  MoveL 5922 to (-205.95, 106.69, -39.37) mm, rotated rx -180 ry 0 rz 0.01 deg; joints [32.683, -45.289, 105.651, -143.751, 66, 164.377]
  MoveL 5923 to (-200.36, 103.18, -39.61) mm, rotated rx 180 ry 0 rz 0.01 deg; joints [32.686, -45.553, 106.254, -143.837, 66.275, 164.595]
  MoveL 5924 to (-194.9, 106.89, -39.86) mm, rotated rx 180 ry 0 rz 0.01 deg; joints [32.922, -45.653, 106.489, -143.624, 66.452, 164.581]
  MoveL 5925 to (-196.11, 113.38, -40.1) mm, rotated rx -180 ry 0 rz 0.01 deg; joints [33.109, -45.453, 106.072, -143.373, 66.332, 164.36]
  MoveL 5926 to (-202.54, 114.87, -40.35) mm, rotated rx 180 ry 0 rz 0.01 deg; joints [33.021, -45.178, 105.502, -143.387, 66.069, 164.205]
  MoveL 5927 to (-206.49, 109.57, -40.59) mm, rotated rx 180 ry 0 rz 0.01 deg; joints [32.766, -45.142, 105.46, -143.652, 65.99, 164.313]
  MoveL 5928 to (-203.21, 103.84, -40.83) mm, rotated rx 180 ry 0 rz 0.01 deg; joints [32.648, -45.372, 105.996, -143.856, 66.202, 164.561]
  MoveL 5929 to (-196.65, 104.54, -41.08) mm, rotated rx -180 ry 0 rz 0.01 deg; joints [32.809, -45.577, 106.465, -143.756, 66.461, 164.662]
  MoveL 5930 to (-194.66, 110.84, -41.32) mm, rotated rx 180 ry 0 rz 0.01 deg; joints [33.057, -45.496, 106.304, -143.476, 66.469, 164.505]
  MoveL 5931 to (-199.63, 115.18, -41.57) mm, rotated rx -180 ry 0 rz 0.01 deg; joints [33.093, -45.21, 105.704, -143.357, 66.227, 164.285]
  MoveL 5932 to (-205.6, 112.37, -41.81) mm, rotated rx -180 ry 0 rz 0.01 deg; joints [32.876, -45.046, 105.383, -143.542, 66.037, 164.276]
  MoveL 5933 to (-205.42, 105.77, -42.05) mm, rotated rx 180 ry 0 rz 0.01 deg; joints [32.666, -45.186, 105.724, -143.815, 66.137, 164.498]
  MoveL 5934 to (-199.3, 103.29, -42.3) mm, rotated rx 180 ry 0 rz 0.01 deg; joints [32.713, -45.445, 106.317, -143.852, 66.42, 164.693]
  MoveL 5935 to (-194.57, 107.91, -42.54) mm, rotated rx 180 ry 0 rz 0.01 deg; joints [32.964, -45.498, 106.449, -143.611, 66.557, 164.637]
  MoveL 5936 to (-196.91, 114.08, -42.79) mm, rotated rx 180 ry 0 rz 0.01 deg; joints [33.116, -45.266, 105.962, -143.386, 66.396, 164.406]
  MoveL 5937 to (-203.51, 114.42, -43.03) mm, rotated rx 180 ry 0 rz 0.01 deg; joints [32.988, -45.011, 105.436, -143.449, 66.141, 164.286]
  MoveL 5938 to (-206.46, 108.51, -43.27) mm, rotated rx 180 ry 0 rz 0.01 deg; joints [32.734, -45.024, 105.501, -143.728, 66.109, 164.43]
  MoveL 5939 to (-202.22, 103.44, -43.52) mm, rotated rx 180 ry 0 rz 0.01 deg; joints [32.657, -45.273, 106.078, -143.893, 66.351, 164.674]
  MoveL 5940 to (-195.88, 105.28, -43.76) mm, rotated rx -180 ry 0 rz 0.01 deg; joints [32.851, -45.444, 106.472, -143.748, 66.587, 164.735]
  MoveL 5941 to (-195.03, 111.83, -44.01) mm, rotated rx 180 ry 0 rz 0.01 deg; joints [33.083, -45.317, 106.211, -143.472, 66.546, 164.549]
  MoveL 5942 to (-200.69, 115.24, -44.25) mm, rotated rx 180 ry 0 rz 0.01 deg; joints [33.074, -45.028, 105.605, -143.399, 66.288, 164.347]
  MoveL 5943 to (-206.08, 111.41, -44.49) mm, rotated rx 180 ry 0 rz 0.01 deg; joints [32.837, -44.908, 105.38, -143.619, 66.134, 164.381]
  MoveL 5944 to (-204.74, 104.95, -44.74) mm, rotated rx -180 ry 0 rz 0.01 deg; joints [32.655, -45.085, 105.803, -143.873, 66.279, 164.619]
  MoveL 5945 to (-198.27, 103.59, -44.98) mm, rotated rx 180 ry 0 rz 0.01 deg; joints [32.746, -45.331, 106.366, -143.86, 66.562, 164.784]
  MoveL 5946 to (-194.44, 108.96, -45.23) mm, rotated rx 180 ry 0 rz 0.01 deg; joints [33.003, -45.335, 106.393, -143.597, 66.654, 164.689]
  MoveL 5947 to (-197.83, 114.63, -45.47) mm, rotated rx 180 ry 0 rz 0.01 deg; joints [33.116, -45.078, 105.849, -143.406, 66.456, 164.456]
  MoveL 5948 to (-204.38, 113.8, -45.71) mm, rotated rx 180 ry 0 rz 0.01 deg; joints [32.951, -44.851, 105.385, -143.516, 66.217, 164.372]
  MoveL 5949 to (-206.24, 107.46, -45.96) mm, rotated rx 180 ry 0 rz 0.01 deg; joints [32.706, -44.912, 105.555, -143.801, 66.235, 164.549]
  MoveL 5950 to (-201.18, 103.22, -46.2) mm, rotated rx 180 ry 0 rz 0.01 deg; joints [32.673, -45.171, 106.154, -143.922, 66.499, 164.782]
  MoveL 5951 to (-195.26, 106.15, -46.45) mm, rotated rx -180 ry 0 rz 0.01 deg; joints [32.894, -45.302, 106.462, -143.737, 66.705, 164.801]
  MoveL 5952 to (-195.58, 112.75, -46.69) mm, rotated rx 180 ry 0 rz 0.01 deg; joints [33.103, -45.133, 106.109, -143.472, 66.616, 164.594]
  MoveL 5953 to (-201.75, 115.1, -46.93) mm, rotated rx -180 ry 0 rz 0.01 deg; joints [33.049, -44.85, 105.516, -143.448, 66.352, 164.415]
  MoveL 5954 to (-206.38, 110.39, -47.18) mm, rotated rx -180 ry 0 rz 0.01 deg; joints [32.799, -44.777, 105.392, -143.696, 66.238, 164.49]
  MoveL 5955 to (-203.92, 104.26, -47.42) mm, rotated rx 180 ry 0 rz 0.01 deg; joints [32.651, -44.986, 105.885, -143.924, 66.425, 164.737]
  MoveL 5956 to (-197.32, 104.06, -47.67) mm, rotated rx 180 ry 0 rz 0.01 deg; joints [32.783, -45.21, 106.401, -143.861, 66.698, 164.868]
  MoveL 5957 to (-194.49, 110.03, -47.91) mm, rotated rx -180 ry 0 rz 0.01 deg; joints [33.038, -45.166, 106.321, -143.585, 66.742, 164.737]
  MoveL 5958 to (-198.82, 115.01, -48.15) mm, rotated rx -180 ry 0 rz 0.01 deg; joints [33.109, -44.891, 105.739, -143.433, 66.516, 164.508]
  MoveL 5959 to (-205.13, 113.04, -48.4) mm, rotated rx -180 ry 0 rz 0.01 deg; joints [32.912, -44.698, 105.35, -143.588, 66.301, 164.466]
  MoveL 5960 to (-205.84, 106.47, -48.64) mm, rotated rx -180 ry 0 rz 0.01 deg; joints [32.683, -44.804, 105.62, -143.869, 66.367, 164.67]
  MoveL 5961 to (-200.11, 103.19, -48.89) mm, rotated rx -180 ry 0 rz 0.01 deg; joints [32.696, -45.065, 106.222, -143.943, 66.646, 164.884]
  MoveL 5962 to (-194.81, 107.12, -49.13) mm, rotated rx -180 ry 0 rz 0.01 deg; joints [32.937, -45.153, 106.434, -143.723, 66.815, 164.861]
  MoveL 5963 to (-196.28, 113.55, -49.38) mm, rotated rx 180 ry 0 rz 0.01 deg; joints [33.116, -44.947, 106, -143.478, 66.682, 164.638]
  MoveL 5964 to (-202.77, 114.78, -49.62) mm, rotated rx 180 ry 0 rz 0.01 deg; joints [33.019, -44.678, 105.438, -143.504, 66.418, 164.49]
  MoveL 5965 to (-206.5, 109.33, -49.86) mm, rotated rx -180 ry 0 rz 0.01 deg; joints [32.763, -44.653, 105.421, -143.773, 66.351, 164.604]
  MoveL 5966 to (-202.99, 103.73, -50.11) mm, rotated rx -180 ry 0 rz 0.01 deg; joints [32.654, -44.886, 105.967, -143.967, 66.572, 164.852]
  MoveL 5967 to (-196.46, 104.7, -50.35) mm, rotated rx 180 ry 0 rz 0.01 deg; joints [32.824, -45.082, 106.42, -143.856, 66.828, 164.946]
  MoveL 5968 to (-194.73, 111.07, -50.6) mm, rotated rx -180 ry 0 rz 0.01 deg; joints [33.069, -44.991, 106.235, -143.577, 66.823, 164.782]
  MoveL 5969 to (-199.87, 115.21, -50.84) mm, rotated rx -180 ry 0 rz 0.01 deg; joints [33.094, -44.706, 105.633, -143.468, 66.575, 164.565]
  MoveL 5970 to (-205.73, 112.16, -51.08) mm, rotated rx -180 ry 0 rz 0.01 deg; joints [32.872, -44.553, 105.332, -143.662, 66.391, 164.565]
  MoveL 5971 to (-205.28, 105.57, -51.33) mm, rotated rx -180 ry 0 rz 0.01 deg; joints [32.667, -44.7, 105.692, -143.931, 66.505, 164.79]
  MoveL 5972 to (-199.06, 103.34, -51.57) mm, rotated rx -180 ry 0 rz 0.01 deg; joints [32.725, -44.954, 106.28, -143.955, 66.791, 164.979]
  MoveL 5973 to (-194.53, 108.15, -51.82) mm, rotated rx -180 ry 0 rz 0.01 deg; joints [32.978, -44.996, 106.389, -143.708, 66.916, 164.916]
  MoveL 5974 to (-197.11, 114.22, -52.06) mm, rotated rx 180 ry 0 rz 0.01 deg; joints [33.121, -44.759, 105.886, -143.492, 66.744, 164.684]
  MoveL 5975 to (-203.72, 114.29, -52.3) mm, rotated rx 180 ry 0 rz 0.01 deg; joints [32.984, -44.512, 105.374, -143.566, 66.49, 164.57]
  MoveL 5976 to (-206.42, 108.27, -52.55) mm, rotated rx 180 ry 0 rz 0.01 deg; joints [32.732, -44.536, 105.463, -143.847, 66.471, 164.721]
  MoveL 5977 to (-201.99, 103.37, -52.79) mm, rotated rx 180 ry 0 rz 0.01 deg; joints [32.665, -44.785, 106.046, -144.001, 66.721, 164.963]
  MoveL 5978 to (-195.73, 105.47, -53.04) mm, rotated rx 180 ry 0 rz 0.01 deg; joints [32.866, -44.946, 106.421, -143.846, 66.951, 165.016]
  MoveL 5979 to (-195.14, 112.05, -53.28) mm, rotated rx 180 ry 0 rz 0.01 deg; joints [33.093, -44.81, 106.138, -143.572, 66.897, 164.826]
  MoveL 5980 to (-200.94, 115.22, -53.52) mm, rotated rx 180 ry 0 rz 0.01 deg; joints [33.074, -44.525, 105.534, -143.511, 66.635, 164.628]
  MoveL 5981 to (-206.16, 111.18, -53.77) mm, rotated rx -180 ry 0 rz 0.01 deg; joints [32.833, -44.416, 105.33, -143.738, 66.489, 164.669]
  MoveL 5982 to (-204.56, 104.78, -54.01) mm, rotated rx 180 ry 0 rz 0.01 deg; joints [32.658, -44.599, 105.77, -143.986, 66.647, 164.909]
  MoveL 5983 to (-198.05, 103.68, -54.26) mm, rotated rx 180 ry 0 rz 0.01 deg; joints [32.759, -44.838, 106.324, -143.96, 66.93, 165.068]
  MoveL 5984 to (-194.43, 109.21, -54.5) mm, rotated rx 180 ry 0 rz 0.01 deg; joints [33.016, -44.831, 106.326, -143.694, 67.01, 164.966]
  MoveC 5985 to (-196.76, 111.53, -54.5) mm, rotated rx 180 ry 0 rz 0.01 deg; joints [33.043, -44.7, 106.033, -143.626, 66.887, 164.85] to (-199.08, 109.21, -54.5) mm, rotated rx -180 ry 0 rz 0.01 deg; joints [32.918, -44.669, 105.97, -143.748, 66.826, 164.882]
  MoveC 5986 to (-196.76, 106.88, -54.5) mm, rotated rx -180 ry 0 rz 0.01 deg; joints [32.891, -44.801, 106.264, -143.817, 66.949, 164.997] to (-194.43, 109.21, -54.5) mm, rotated rx -180 ry 0 rz 0.01 deg; joints [33.016, -44.831, 106.326, -143.694, 67.01, 164.966]
  MoveC 5987 to (-193.87, 111.26, -54.5) mm, rotated rx 180 ry 0 rz 0.01 deg; joints [33.095, -44.806, 106.268, -143.604, 67.005, 164.911] to (-192.35, 112.73, -54.5) mm, rotated rx -180 ry 0 rz 0.01 deg; joints [33.176, -44.827, 106.311, -143.526, 67.046, 164.892]
  MoveC 5988 to (-191.13, 114.78, -54.5) mm, rotated rx -180 ry 0 rz 0.01 deg; joints [33.268, -44.825, 106.301, -143.428, 67.066, 164.849] to (-192.33, 116.83, -54.5) mm, rotated rx 180 ry 0 rz 0.01 deg; joints [33.309, -44.738, 106.107, -143.358, 66.992, 164.762]
  MoveC 5989 to (-193.08, 117.28, -54.5) mm, rotated rx -180 ry 0 rz 0.01 deg; joints [33.308, -44.702, 106.027, -143.348, 66.956, 164.734] to (-193.81, 117.76, -54.5) mm, rotated rx 180 ry 0 rz 0.01 deg; joints [33.308, -44.666, 105.947, -143.337, 66.921, 164.705]
  MoveC 5990 to (-196.76, 118.7, -54.5) mm, rotated rx 180 ry 0 rz 0.01 deg; joints [33.275, -44.542, 105.675, -143.332, 66.792, 164.622] to (-199.7, 117.76, -54.5) mm, rotated rx 180 ry 0 rz 0.01 deg; joints [33.183, -44.46, 105.496, -143.404, 66.688, 164.599]
  MoveC 5991 to (-201.1, 116.87, -54.5) mm, rotated rx 180 ry 0 rz 0.01 deg; joints [33.124, -44.43, 105.432, -143.456, 66.644, 164.602] to (-202.59, 116.12, -54.5) mm, rotated rx -180 ry 0 rz 0.01 deg; joints [33.069, -44.394, 105.355, -143.504, 66.595, 164.599]
  MoveC 5992 to (-204.95, 114.01, -54.5) mm, rotated rx 180 ry 0 rz 0.01 deg; joints [32.951, -44.358, 105.279, -143.617, 66.529, 164.623] to (-205.64, 110.92, -54.5) mm, rotated rx -180 ry 0 rz 0.01 deg; joints [32.836, -44.401, 105.38, -143.751, 66.542, 164.709]
  MoveC 5993 to (-205.56, 109.27, -54.5) mm, rotated rx -180 ry 0 rz 0.01 deg; joints [32.784, -44.44, 105.467, -143.819, 66.567, 164.763] to (-205.65, 107.61, -54.5) mm, rotated rx 180 ry 0 rz 0.01 deg; joints [32.728, -44.473, 105.543, -143.888, 66.585, 164.814]
  MoveC 5994 to (-205, 104.51, -54.5) mm, rotated rx 180 ry 0 rz 0.01 deg; joints [32.64, -44.563, 105.747, -144.008, 66.652, 164.924] to (-202.66, 102.37, -54.5) mm, rotated rx -180 ry 0 rz 0.01 deg; joints [32.619, -44.691, 106.032, -144.07, 66.773, 165.034]
  MoveC 5995 to (-201.23, 101.62, -54.5) mm, rotated rx -180 ry 0 rz 0.01 deg; joints [32.625, -44.758, 106.18, -144.084, 66.841, 165.083] to (-199.87, 100.74, -54.5) mm, rotated rx -180 ry 0 rz 0.01 deg; joints [32.624, -44.824, 106.328, -144.105, 66.906, 165.135]
  MoveC 5996 to (-196.86, 99.74, -54.5) mm, rotated rx -180 ry 0 rz 0.01 deg; joints [32.655, -44.951, 106.608, -144.112, 67.039, 165.22] to (-193.81, 100.62, -54.5) mm, rotated rx -180 ry 0 rz 0.01 deg; joints [32.748, -45.038, 106.797, -144.04, 67.148, 165.247]
  MoveC 5997 to (-193.08, 101.1, -54.5) mm, rotated rx 180 ry 0 rz 0.01 deg; joints [32.779, -45.053, 106.83, -144.011, 67.171, 165.245] to (-192.33, 101.56, -54.5) mm, rotated rx -180 ry 0 rz 0.01 deg; joints [32.81, -45.069, 106.864, -143.984, 67.194, 165.244]
  MoveC 5998 to (-191.57, 102, -54.5) mm, rotated rx -180 ry 0 rz 0.01 deg; joints [32.841, -45.086, 106.901, -143.957, 67.219, 165.244] to (-190.79, 102.39, -54.5) mm, rotated rx -180 ry 0 rz 0.01 deg; joints [32.87, -45.105, 106.941, -143.931, 67.244, 165.245]
  MoveC 5999 to (-188.5, 104.54, -54.5) mm, rotated rx -180 ry 0 rz 0.01 deg; joints [32.99, -45.138, 107.011, -143.816, 67.306, 165.219] to (-187.86, 107.61, -54.5) mm, rotated rx -180 ry 0 rz 0.01 deg; joints [33.104, -45.094, 106.907, -143.682, 67.291, 165.134]
  MoveC 6000 to (-187.95, 109.27, -54.5) mm, rotated rx 180 ry 0 rz 0.01 deg; joints [33.156, -45.055, 106.819, -143.616, 67.265, 165.08] to (-187.87, 110.92, -54.5) mm, rotated rx 180 ry 0 rz 0.01 deg; joints [33.212, -45.022, 106.742, -143.547, 67.246, 165.029]
  MoveC 6001 to (-188.56, 114.01, -54.5) mm, rotated rx 180 ry 0 rz 0.01 deg; joints [33.298, -44.931, 106.535, -143.429, 67.178, 164.919] to (-190.92, 116.12, -54.5) mm, rotated rx 180 ry 0 rz 0.01 deg; joints [33.316, -44.802, 106.25, -143.37, 67.057, 164.81]
  MoveC 6002 to (-191.64, 116.46, -54.5) mm, rotated rx 180 ry 0 rz 0.01 deg; joints [33.312, -44.77, 106.179, -143.365, 67.024, 164.786] to (-192.33, 116.83, -54.5) mm, rotated rx 180 ry 0 rz 0.01 deg; joints [33.309, -44.738, 106.107, -143.358, 66.992, 164.762]
  MoveL 6003 to (-192.94, 116.99, -54.33) mm, rotated rx 180 ry 0 rz 0.01 deg; joints [33.301, -44.722, 106.054, -143.356, 66.959, 164.741]
  MoveL 6004 to (-193.39, 116.91, -53.87) mm, rotated rx -180 ry 0 rz 0.01 deg; joints [33.289, -44.733, 106.026, -143.359, 66.924, 164.721]
  MoveL 6005 to (-193.55, 116.84, -53.23) mm, rotated rx 180 ry 0 rz 0.01 deg; joints [33.283, -44.764, 106.021, -143.357, 66.895, 164.701]
  Set speed (500.0 mm/s)
  MoveL 6006 to (-193.55, 116.84, 11) mm, rotated rx 180 ry 0 rz 0.01 deg; joints [33.247, -48.144, 106.249, -142.533, 64.368, 162.631]
  Set speed (500.0 mm/s)
  MoveL 6007 to (-195.99, 9.53, 11) mm, rotated rx -180 ry 0 rz 0.01 deg; joints [29.569, -50.402, 111.086, -147.114, 65.397, 165.962]
  Set speed (500.0 mm/s)
  MoveL 6008 to (-195.99, 9.53, -32.73) mm, rotated rx 180 ry 0 rz 0.01 deg; joints [29.597, -48.003, 110.965, -147.623, 67.321, 167.29]
  Set speed (100.0 mm/s)
  MoveL 6009 to (-196.15, 9.55, -33.35) mm, rotated rx 180 ry 0 rz 0.01 deg; joints [29.595, -47.963, 110.949, -147.63, 67.342, 167.305]
  MoveL 6010 to (-196.6, 9.58, -33.82) mm, rotated rx 180 ry 0 rz 0.01 deg; joints [29.587, -47.921, 110.911, -147.639, 67.344, 167.311]
  MoveL 6011 to (-197.22, 9.56, -34) mm, rotated rx -180 ry 0 rz 0.01 deg; joints [29.574, -47.889, 110.864, -147.649, 67.327, 167.307]
  MoveL 6012 to (-202.45, 5.54, -34.24) mm, rotated rx -180 ry 0 rz 0.01 deg; joints [29.33, -47.766, 110.634, -147.882, 67.177, 167.348]
  MoveL 6013 to (-200.86, -0.87, -34.49) mm, rotated rx 180 ry 0 rz 0.01 deg; joints [29.136, -47.93, 111.031, -148.138, 67.329, 167.563]
  MoveL 6014 to (-194.35, -1.99, -34.73) mm, rotated rx 180 ry 0 rz 0.01 deg; joints [29.225, -48.167, 111.578, -148.112, 67.613, 167.703]
  MoveL 6015 to (-190.73, 3.53, -34.98) mm, rotated rx 180 ry 0 rz 0.01 deg; joints [29.492, -48.177, 111.617, -147.838, 67.701, 167.61]
  MoveL 6016 to (-194.33, 9.07, -35.22) mm, rotated rx 180 ry 0 rz 0.01 deg; joints [29.615, -47.932, 111.101, -147.649, 67.501, 167.403]
  MoveL 6017 to (-200.84, 7.98, -35.46) mm, rotated rx -180 ry 0 rz 0.01 deg; joints [29.448, -47.709, 110.646, -147.773, 67.265, 167.338]
  MoveL 6018 to (-202.46, 1.58, -35.71) mm, rotated rx -180 ry 0 rz 0.01 deg; joints [29.192, -47.759, 110.797, -148.066, 67.288, 167.503]
  MoveL 6019 to (-197.25, -2.47, -35.95) mm, rotated rx 180 ry 0 rz 0.01 deg; joints [29.152, -48.006, 111.371, -148.179, 67.557, 167.707]
  MoveL 6020 to (-191.44, 0.69, -36.2) mm, rotated rx 180 ry 0 rz 0.01 deg; joints [29.378, -48.137, 111.679, -147.98, 67.76, 167.715]
  MoveL 6021 to (-192.01, 7.27, -36.44) mm, rotated rx -180 ry 0 rz 0.01 deg; joints [29.599, -47.979, 111.35, -147.711, 67.668, 167.526]
  MoveL 6022 to (-198.27, 9.39, -36.68) mm, rotated rx 180 ry 0 rz 0.01 deg; joints [29.549, -47.706, 110.777, -147.697, 67.403, 167.374]
  MoveL 6023 to (-202.71, 4.5, -36.93) mm, rotated rx -180 ry 0 rz 0.01 deg; joints [29.29, -47.627, 110.646, -147.958, 67.295, 167.451]
  MoveL 6024 to (-200.02, -1.53, -37.17) mm, rotated rx -180 ry 0 rz 0.01 deg; joints [29.131, -47.822, 111.111, -148.185, 67.487, 167.672]
  MoveL 6025 to (-193.42, -1.48, -37.42) mm, rotated rx 180 ry 0 rz 0.01 deg; joints [29.263, -48.04, 111.615, -148.108, 67.761, 167.781]
  MoveL 6026 to (-190.82, 4.59, -37.66) mm, rotated rx -180 ry 0 rz 0.01 deg; joints [29.53, -48.003, 111.551, -147.822, 67.801, 167.657]
  MoveL 6027 to (-195.34, 9.41, -37.9) mm, rotated rx 180 ry 0 rz 0.01 deg; joints [29.609, -47.74, 110.995, -147.675, 67.572, 167.455]
  MoveL 6028 to (-201.56, 7.2, -38.15) mm, rotated rx -180 ry 0 rz 0.01 deg; joints [29.408, -47.549, 110.612, -147.844, 67.361, 167.427]
  MoveL 6029 to (-202.03, 0.61, -38.39) mm, rotated rx -180 ry 0 rz 0.01 deg; joints [29.168, -47.643, 110.859, -148.13, 67.433, 167.615]
  MoveL 6030 to (-196.18, -2.46, -38.64) mm, rotated rx -180 ry 0 rz 0.01 deg; joints [29.175, -47.893, 111.439, -148.195, 67.716, 167.801]
  MoveL 6031 to (-191.02, 1.67, -38.88) mm, rotated rx 180 ry 0 rz 0.01 deg; joints [29.423, -47.982, 111.655, -147.961, 67.882, 167.772]
  MoveL 6032 to (-192.74, 8.05, -39.13) mm, rotated rx 180 ry 0 rz 0.01 deg; joints [29.614, -47.789, 111.247, -147.715, 67.745, 167.571]
  MoveL 6033 to (-199.27, 9.03, -39.37) mm, rotated rx 180 ry 0 rz 0.01 deg; joints [29.518, -47.527, 110.702, -147.753, 67.483, 167.446]
  MoveL 6034 to (-202.79, 3.44, -39.61) mm, rotated rx -180 ry 0 rz 0.01 deg; joints [29.253, -47.495, 110.672, -148.032, 67.421, 167.557]
  MoveL 6035 to (-199.08, -2.02, -39.86) mm, rotated rx 180 ry 0 rz 0.01 deg; joints [29.134, -47.714, 111.191, -148.223, 67.648, 167.778]
  MoveL 6036 to (-192.58, -0.81, -40.1) mm, rotated rx -180 ry 0 rz 0.01 deg; joints [29.305, -47.905, 111.636, -148.097, 67.903, 167.853]
  MoveL 6037 to (-191.09, 5.62, -40.35) mm, rotated rx -180 ry 0 rz 0.01 deg; joints [29.562, -47.823, 111.472, -147.81, 67.894, 167.701]
  MoveL 6038 to (-196.39, 9.57, -40.59) mm, rotated rx -180 ry 0 rz 0.01 deg; joints [29.595, -47.55, 110.894, -147.709, 67.644, 167.512]
  MoveL 6039 to (-202.13, 6.29, -40.83) mm, rotated rx -180 ry 0 rz 0.01 deg; joints [29.367, -47.397, 110.593, -147.916, 67.465, 167.522]
  MoveL 6040 to (-201.43, -0.27, -41.08) mm, rotated rx -180 ry 0 rz 0.01 deg; joints [29.15, -47.531, 110.929, -148.188, 67.584, 167.726]
  MoveL 6041 to (-195.13, -2.26, -41.32) mm, rotated rx -180 ry 0 rz 0.01 deg; joints [29.204, -47.775, 111.497, -148.202, 67.872, 167.889]
  MoveL 6042 to (-190.78, 2.71, -41.57) mm, rotated rx -180 ry 0 rz 0.01 deg; joints [29.466, -47.82, 111.615, -147.942, 67.995, 167.824]
  MoveL 6043 to (-193.6, 8.68, -41.81) mm, rotated rx 180 ry 0 rz 0.01 deg; joints [29.621, -47.596, 111.14, -147.726, 67.819, 167.617]
  MoveL 6044 to (-200.2, 8.5, -42.05) mm, rotated rx -180 ry 0 rz 0.01 deg; joints [29.483, -47.355, 110.64, -147.814, 67.567, 167.524]
  MoveL 6045 to (-202.68, 2.38, -42.3) mm, rotated rx -180 ry 0 rz 0.01 deg; joints [29.22, -47.369, 110.712, -148.103, 67.554, 167.666]
  MoveL 6046 to (-198.06, -2.35, -42.54) mm, rotated rx 180 ry 0 rz 0.01 deg; joints [29.144, -47.605, 111.269, -148.252, 67.809, 167.88]
  MoveL 6047 to (-191.88, -0.01, -42.79) mm, rotated rx -180 ry 0 rz 0.01 deg; joints [29.349, -47.764, 111.641, -148.083, 68.038, 167.919]
  MoveL 6048 to (-191.55, 6.59, -43.03) mm, rotated rx -180 ry 0 rz 0.01 deg; joints [29.589, -47.639, 111.381, -147.803, 67.98, 167.745]
  MoveL 6049 to (-197.46, 9.54, -43.27) mm, rotated rx 180 ry 0 rz 0.01 deg; joints [29.575, -47.363, 110.799, -147.751, 67.717, 167.574]
  MoveL 6050 to (-202.53, 5.3, -43.52) mm, rotated rx 180 ry 0 rz 0.01 deg; joints [29.326, -47.252, 110.591, -147.991, 67.576, 167.62]
  MoveL 6051 to (-200.68, -1.04, -43.76) mm, rotated rx -180 ry 0 rz 0.01 deg; joints [29.14, -47.421, 111.005, -148.24, 67.74, 167.837]
  MoveL 6052 to (-194.13, -1.89, -44.01) mm, rotated rx 180 ry 0 rz 0.01 deg; joints [29.239, -47.651, 111.543, -148.201, 68.024, 167.971]
  MoveL 6053 to (-190.73, 3.77, -44.25) mm, rotated rx 180 ry 0 rz 0.01 deg; joints [29.507, -47.651, 111.559, -147.924, 68.1, 167.873]
  MoveL 6054 to (-194.55, 9.16, -44.49) mm, rotated rx 180 ry 0 rz 0.01 deg; joints [29.62, -47.403, 111.032, -147.745, 67.89, 167.666]
  MoveL 6055 to (-201.02, 7.82, -44.74) mm, rotated rx 180 ry 0 rz 0.01 deg; joints [29.445, -47.189, 110.592, -147.88, 67.658, 167.608]
  MoveL 6056 to (-202.38, 1.35, -44.98) mm, rotated rx -180 ry 0 rz 0.01 deg; joints [29.191, -47.249, 110.765, -148.171, 67.694, 167.777]
  MoveL 6057 to (-197, -2.48, -45.23) mm, rotated rx -180 ry 0 rz 0.01 deg; joints [29.162, -47.494, 111.342, -148.273, 67.969, 167.977]
  MoveL 6058 to (-191.33, 0.91, -45.47) mm, rotated rx -180 ry 0 rz 0.01 deg; joints [29.394, -47.614, 111.629, -148.065, 68.165, 167.979]
  MoveL 6059 to (-192.17, 7.46, -45.71) mm, rotated rx -180 ry 0 rz 0.01 deg; joints [29.609, -47.45, 111.281, -147.801, 68.06, 167.788]
  MoveL 6060 to (-198.5, 9.32, -45.96) mm, rotated rx -180 ry 0 rz 0.01 deg; joints [29.548, -47.181, 110.713, -147.8, 67.792, 167.64]
  MoveL 6061 to (-202.75, 4.26, -46.2) mm, rotated rx -180 ry 0 rz 0.01 deg; joints [29.287, -47.113, 110.604, -148.065, 67.695, 167.723]
  MoveL 6062 to (-199.81, -1.66, -46.45) mm, rotated rx -180 ry 0 rz 0.01 deg; joints [29.137, -47.312, 111.083, -148.283, 67.898, 167.944]
  MoveL 6063 to (-193.22, -1.34, -46.69) mm, rotated rx 180 ry 0 rz 0.01 deg; joints [29.278, -47.521, 111.574, -148.194, 68.171, 168.047]
  MoveL 6064 to (-190.86, 4.83, -46.93) mm, rotated rx -180 ry 0 rz 0.01 deg; joints [29.543, -47.475, 111.488, -147.908, 68.198, 167.918]
  MoveL 6065 to (-195.58, 9.46, -47.18) mm, rotated rx -180 ry 0 rz 0.01 deg; joints [29.612, -47.212, 110.925, -147.772, 67.96, 167.719]
  MoveL 6066 to (-201.7, 7, -47.42) mm, rotated rx -180 ry 0 rz 0.01 deg; joints [29.404, -47.03, 110.559, -147.95, 67.755, 167.697]
  MoveL 6067 to (-201.9, 0.4, -47.67) mm, rotated rx 180 ry 0 rz 0.01 deg; joints [29.169, -47.132, 110.827, -148.233, 67.841, 167.888]
  MoveL 6068 to (-195.94, -2.43, -47.91) mm, rotated rx 180 ry 0 rz 0.01 deg; joints [29.186, -47.378, 111.406, -148.285, 68.128, 168.069]
  MoveL 6069 to (-190.95, 1.9, -48.15) mm, rotated rx -180 ry 0 rz 0.01 deg; joints [29.439, -47.457, 111.6, -148.045, 68.284, 168.034]
  MoveL 6070 to (-192.93, 8.21, -48.4) mm, rotated rx -180 ry 0 rz 0.01 deg; joints [29.621, -47.258, 111.175, -147.806, 68.135, 167.832]
  MoveL 6071 to (-199.49, 8.92, -48.64) mm, rotated rx -180 ry 0 rz 0.01 deg; joints [29.516, -47.003, 110.639, -147.856, 67.872, 167.713]
  MoveL 6072 to (-202.78, 3.19, -48.89) mm, rotated rx 180 ry 0 rz 0.01 deg; joints [29.25, -46.982, 110.632, -148.138, 67.822, 167.829]
  MoveL 6073 to (-198.85, -2.11, -49.13) mm, rotated rx 180 ry 0 rz 0.01 deg; joints [29.141, -47.203, 111.161, -148.318, 68.059, 168.048]
  MoveL 6074 to (-192.41, -0.64, -49.37) mm, rotated rx 180 ry 0 rz 0.01 deg; joints [29.321, -47.385, 111.59, -148.182, 68.31, 168.117]
  MoveL 6075 to (-191.18, 5.85, -49.62) mm, rotated rx 180 ry 0 rz 0.01 deg; joints [29.574, -47.293, 111.403, -147.896, 68.287, 167.961]
  MoveL 6076 to (-196.64, 9.58, -49.86) mm, rotated rx 180 ry 0 rz 0.01 deg; joints [29.596, -47.022, 110.823, -147.807, 68.031, 167.775]
  MoveL 6077 to (-202.24, 6.07, -50.11) mm, rotated rx 180 ry 0 rz 0.01 deg; joints [29.363, -46.879, 110.543, -148.022, 67.86, 167.791]
  MoveL 6078 to (-201.27, -0.46, -50.35) mm, rotated rx 180 ry 0 rz 0.01 deg; joints [29.153, -47.019, 110.897, -148.289, 67.992, 167.998]
  MoveL 6079 to (-194.9, -2.19, -50.6) mm, rotated rx -180 ry 0 rz 0.01 deg; joints [29.217, -47.258, 111.459, -148.289, 68.283, 168.155]
  MoveL 6080 to (-190.75, 2.95, -50.84) mm, rotated rx 180 ry 0 rz 0.01 deg; joints [29.481, -47.293, 111.554, -148.025, 68.394, 168.084]
  MoveL 6081 to (-193.81, 8.81, -51.08) mm, rotated rx 180 ry 0 rz 0.01 deg; joints [29.627, -47.065, 111.066, -147.818, 68.207, 167.877]
  MoveL 6082 to (-200.4, 8.36, -51.33) mm, rotated rx -180 ry 0 rz 0.01 deg; joints [29.48, -46.832, 110.578, -147.917, 67.957, 167.791]
  MoveL 6083 to (-202.62, 2.14, -51.57) mm, rotated rx -180 ry 0 rz 0.01 deg; joints [29.218, -46.856, 110.673, -148.207, 67.957, 167.937]
  MoveL 6084 to (-197.82, -2.39, -51.82) mm, rotated rx 180 ry 0 rz 0.01 deg; joints [29.153, -47.092, 111.236, -148.345, 68.219, 168.149]
  MoveL 6085 to (-191.74, 0.19, -52.06) mm, rotated rx -180 ry 0 rz 0.01 deg; joints [29.365, -47.24, 111.59, -148.166, 68.442, 168.181]
  MoveL 6086 to (-191.68, 6.8, -52.3) mm, rotated rx 180 ry 0 rz 0.01 deg; joints [29.599, -47.107, 111.308, -147.889, 68.371, 168.003]
  MoveL 6087 to (-197.7, 9.5, -52.55) mm, rotated rx 180 ry 0 rz 0.01 deg; joints [29.574, -46.835, 110.728, -147.85, 68.103, 167.837]
  MoveL 6088 to (-202.59, 5.07, -52.79) mm, rotated rx 180 ry 0 rz 0.01 deg; joints [29.322, -46.734, 110.542, -148.096, 67.972, 167.89]
  MoveL 6089 to (-200.49, -1.19, -53.04) mm, rotated rx 180 ry 0 rz 0.01 deg; joints [29.144, -46.909, 110.971, -148.337, 68.148, 168.106]
  MoveL 6090 to (-193.92, -1.78, -53.28) mm, rotated rx -180 ry 0 rz 0.01 deg; joints [29.253, -47.132, 111.5, -148.287, 68.432, 168.235]
  MoveL 6091 to (-190.74, 4.02, -53.52) mm, rotated rx 180 ry 0 rz 0.01 deg; joints [29.521, -47.121, 111.492, -148.007, 68.496, 168.131]
  MoveL 6092 to (-194.78, 9.24, -53.77) mm, rotated rx -180 ry 0 rz 0.01 deg; joints [29.624, -46.872, 110.955, -147.838, 68.276, 167.926]
  MoveL 6093 to (-201.19, 7.64, -54.01) mm, rotated rx -180 ry 0 rz 0.01 deg; joints [29.441, -46.667, 110.531, -147.984, 68.048, 167.874]
  MoveL 6094 to (-202.29, 1.13, -54.26) mm, rotated rx 180 ry 0 rz 0.01 deg; joints [29.191, -46.735, 110.726, -148.273, 68.098, 168.047]
  MoveL 6095 to (-196.76, -2.49, -54.5) mm, rotated rx 180 ry 0 rz 0.01 deg; joints [29.172, -46.978, 111.305, -148.362, 68.379, 168.244]
  MoveL 6096 to (-193.31, -2.49, -54.5) mm, rotated rx 180 ry 0 rz 0.01 deg; joints [29.241, -47.097, 111.57, -148.321, 68.519, 168.299]
  MoveC 6097 to (-191.94, -1.39, -54.5) mm, rotated rx 180 ry 0 rz 0.01 deg; joints [29.307, -47.124, 111.627, -148.259, 68.56, 168.291] to (-192.73, 0.17, -54.5) mm, rotated rx 180 ry 0 rz 0.01 deg; joints [29.346, -47.068, 111.499, -148.202, 68.508, 168.234]
  MoveC 6098 to (-193.49, 0.52, -54.5) mm, rotated rx -180 ry 0 rz 0.01 deg; joints [29.343, -47.036, 111.426, -148.197, 68.472, 168.212] to (-194.25, 0.88, -54.5) mm, rotated rx -180 ry 0 rz 0.01 deg; joints [29.341, -47.003, 111.353, -148.191, 68.437, 168.19]
  MoveC 6099 to (-195, 1.24, -54.5) mm, rotated rx 180 ry 0 rz 0.01 deg; joints [29.339, -46.971, 111.279, -148.184, 68.402, 168.168] to (-195.75, 1.63, -54.5) mm, rotated rx 180 ry 0 rz 0.01 deg; joints [29.338, -46.938, 111.206, -148.177, 68.367, 168.145]
  MoveC 6100 to (-196.77, 1.89, -54.5) mm, rotated rx -180 ry 0 rz 0.01 deg; joints [29.327, -46.898, 111.116, -148.178, 68.322, 168.121] to (-197.8, 1.62, -54.5) mm, rotated rx 180 ry 0 rz 0.01 deg; joints [29.297, -46.867, 111.049, -148.202, 68.284, 168.112]
  MoveC 6101 to (-198.51, 1.23, -54.5) mm, rotated rx -180 ry 0 rz 0.01 deg; joints [29.269, -46.85, 111.011, -148.226, 68.26, 168.112] to (-199.22, 0.86, -54.5) mm, rotated rx 180 ry 0 rz 0.01 deg; joints [29.242, -46.832, 110.972, -148.25, 68.236, 168.11]
  MoveC 6102 to (-199.95, 0.51, -54.5) mm, rotated rx 180 ry 0 rz 0.01 deg; joints [29.215, -46.814, 110.931, -148.274, 68.211, 168.109] to (-200.68, 0.17, -54.5) mm, rotated rx -180 ry 0 rz 0.01 deg; joints [29.189, -46.795, 110.889, -148.297, 68.186, 168.106]
  MoveC 6103 to (-201.47, -1.39, -54.5) mm, rotated rx 180 ry 0 rz 0.01 deg; joints [29.119, -46.796, 110.896, -148.371, 68.174, 168.137] to (-200.11, -2.49, -54.5) mm, rotated rx 180 ry 0 rz 0.01 deg; joints [29.107, -46.863, 111.047, -148.402, 68.243, 168.19]
  MoveL 6104 to (-196.76, -2.49, -54.5) mm, rotated rx 180 ry 0 rz 0.01 deg; joints [29.172, -46.978, 111.305, -148.362, 68.379, 168.244]
  MoveC 6105 to (-194.7, -3.11, -54.5) mm, rotated rx 180 ry 0 rz 0.01 deg; joints [29.191, -47.06, 111.489, -148.364, 68.47, 168.294] to (-193.34, -4.77, -54.5) mm, rotated rx -180 ry 0 rz 0.01 deg; joints [29.159, -47.137, 111.664, -148.418, 68.547, 168.362]
  MoveC 6106 to (-191.97, -6.42, -54.5) mm, rotated rx -180 ry 0 rz 0.01 deg; joints [29.128, -47.214, 111.839, -148.471, 68.624, 168.43] to (-189.92, -7.05, -54.5) mm, rotated rx -180 ry 0 rz 0.01 deg; joints [29.146, -47.295, 112.023, -148.472, 68.715, 168.48]
  MoveL 6107 to (-172.14, -7.05, -54.5) mm, rotated rx 180 ry 0 rz 0.01 deg; joints [29.502, -47.898, 113.372, -148.25, 69.429, 168.763]
  MoveC 6108 to (-170.78, -5.95, -54.5) mm, rotated rx -180 ry 0 rz 0.01 deg; joints [29.569, -47.924, 113.428, -148.186, 69.469, 168.754] to (-171.57, -4.39, -54.5) mm, rotated rx 180 ry 0 rz 0.01 deg; joints [29.609, -47.869, 113.302, -148.131, 69.417, 168.699]
  MoveC 6109 to (-177.27, -1.88, -54.5) mm, rotated rx -180 ry 0 rz 0.01 deg; joints [29.583, -47.632, 112.764, -148.098, 69.156, 168.539] to (-183.02, 0.52, -54.5) mm, rotated rx 180 ry 0 rz 0.01 deg; joints [29.552, -47.393, 112.225, -148.069, 68.894, 168.381]
  MoveC 6110 to (-188.71, 3.06, -54.5) mm, rotated rx 180 ry 0 rz 0.01 deg; joints [29.528, -47.153, 111.682, -148.032, 68.632, 168.218] to (-194.21, 6, -54.5) mm, rotated rx 180 ry 0 rz 0.01 deg; joints [29.522, -46.91, 111.135, -147.975, 68.373, 168.047]
  MoveC 6111 to (-196.81, 6.69, -54.5) mm, rotated rx -180 ry 0 rz 0.01 deg; joints [29.495, -46.808, 110.906, -147.977, 68.258, 167.986] to (-199.4, 5.96, -54.5) mm, rotated rx -180 ry 0 rz 0.01 deg; joints [29.418, -46.732, 110.738, -148.038, 68.163, 167.964]
  MoveC 6112 to (-204.83, 2.98, -54.5) mm, rotated rx -180 ry 0 rz 0.01 deg; joints [29.206, -46.599, 110.449, -148.226, 67.981, 167.96] to (-210.48, 0.46, -54.5) mm, rotated rx 180 ry 0 rz 0.01 deg; joints [29.007, -46.449, 110.12, -148.397, 67.783, 167.94]
  MoveC 6113 to (-216.2, -1.9, -54.5) mm, rotated rx 180 ry 0 rz 0.01 deg; joints [28.814, -46.292, 109.777, -148.56, 67.579, 167.914] to (-221.86, -4.39, -54.5) mm, rotated rx 180 ry 0 rz 0.01 deg; joints [28.618, -46.138, 109.44, -148.727, 67.378, 167.892]
  MoveC 6114 to (-222.65, -5.95, -54.5) mm, rotated rx -180 ry 0 rz 0.01 deg; joints [28.549, -46.139, 109.445, -148.801, 67.365, 167.923] to (-221.29, -7.05, -54.5) mm, rotated rx 180 ry 0 rz 0.01 deg; joints [28.536, -46.207, 109.598, -148.833, 67.435, 167.976]
  MoveL 6115 to (-189.92, -7.05, -54.5) mm, rotated rx -180 ry 0 rz 0.01 deg; joints [29.146, -47.295, 112.023, -148.472, 68.715, 168.48]
  MoveC 6116 to (-187.09, -7.9, -54.5) mm, rotated rx 180 ry 0 rz 0.01 deg; joints [29.172, -47.408, 112.275, -148.474, 68.84, 168.549] to (-185.2, -10.19, -54.5) mm, rotated rx -180 ry 0 rz 0.01 deg; joints [29.128, -47.513, 112.516, -148.547, 68.946, 168.641]
  MoveC 6117 to (-183.32, -12.48, -54.5) mm, rotated rx -180 ry 0 rz 0.01 deg; joints [29.084, -47.617, 112.755, -148.621, 69.051, 168.734] to (-180.49, -13.33, -54.5) mm, rotated rx 180 ry 0 rz 0.01 deg; joints [29.109, -47.729, 113.007, -148.622, 69.176, 168.802]
  MoveL 6118 to (-142.96, -13.33, -54.5) mm, rotated rx 180 ry 0 rz 0.01 deg; joints [29.876, -48.975, 115.817, -148.123, 70.671, 169.393]
  MoveC 6119 to (-141.6, -12.24, -54.5) mm, rotated rx 180 ry 0 rz 0.01 deg; joints [29.945, -49, 115.871, -148.058, 70.71, 169.385] to (-142.38, -10.67, -54.5) mm, rotated rx 180 ry 0 rz 0.01 deg; joints [29.985, -48.947, 115.747, -148.003, 70.658, 169.331]
  MoveL 6120 to (-189.17, 10.28, -54.5) mm, rotated rx 180 ry 0 rz 0.01 deg; joints [29.773, -47.004, 111.334, -147.734, 68.52, 168.009]
  MoveC 6121 to (-190.36, 10.9, -54.5) mm, rotated rx 180 ry 0 rz 0.01 deg; joints [29.771, -46.952, 111.217, -147.723, 68.464, 167.972] to (-191.49, 11.62, -54.5) mm, rotated rx -180 ry 0 rz 0.01 deg; joints [29.774, -46.9, 111.099, -147.706, 68.41, 167.933]
  MoveC 6122 to (-192.57, 12.41, -54.5) mm, rotated rx 180 ry 0 rz 0.01 deg; joints [29.78, -46.848, 110.982, -147.686, 68.356, 167.893] to (-193.65, 13.2, -54.5) mm, rotated rx 180 ry 0 rz 0.01 deg; joints [29.786, -46.796, 110.865, -147.666, 68.302, 167.853]
  MoveC 6123 to (-196.68, 14.21, -54.5) mm, rotated rx 180 ry 0 rz 0.01 deg; joints [29.761, -46.673, 110.589, -147.66, 68.167, 167.775] to (-199.72, 13.27, -54.5) mm, rotated rx -180 ry 0 rz 0.01 deg; joints [29.667, -46.585, 110.396, -147.735, 68.056, 167.752]
  MoveC 6124 to (-200.96, 12.4, -54.5) mm, rotated rx 180 ry 0 rz 0.01 deg; joints [29.612, -46.559, 110.339, -147.786, 68.017, 167.757] to (-202.19, 11.52, -54.5) mm, rotated rx -180 ry 0 rz 0.01 deg; joints [29.557, -46.533, 110.283, -147.837, 67.979, 167.762]
  MoveC 6125 to (-203.46, 10.7, -54.5) mm, rotated rx -180 ry 0 rz 0.01 deg; joints [29.503, -46.504, 110.221, -147.887, 67.938, 167.764] to (-204.81, 10, -54.5) mm, rotated rx -180 ry 0 rz 0.01 deg; joints [29.452, -46.47, 110.147, -147.931, 67.892, 167.762]
  MoveL 6126 to (-251.08, -10.67, -54.5) mm, rotated rx -180 ry 0 rz 0.01 deg; joints [27.853, -45.208, 107.395, -149.291, 66.242, 167.595]
  MoveC 6127 to (-251.87, -12.24, -54.5) mm, rotated rx 180 ry 0 rz 0.01 deg; joints [27.784, -45.207, 107.398, -149.364, 66.228, 167.626] to (-250.51, -13.33, -54.5) mm, rotated rx -180 ry 0 rz 0.01 deg; joints [27.771, -45.277, 107.553, -149.398, 66.298, 167.68]
  MoveL 6128 to (-180.49, -13.33, -54.5) mm, rotated rx 180 ry 0 rz 0.01 deg; joints [29.109, -47.729, 113.007, -148.622, 69.176, 168.802]
  MoveC 6129 to (-177.65, -14.19, -54.5) mm, rotated rx 180 ry 0 rz 0.01 deg; joints [29.135, -47.84, 113.258, -148.622, 69.302, 168.87] to (-175.77, -16.48, -54.5) mm, rotated rx -180 ry 0 rz 0.01 deg; joints [29.091, -47.944, 113.496, -148.695, 69.407, 168.962]
  MoveC 6130 to (-173.89, -18.76, -54.5) mm, rotated rx -180 ry 0 rz 0.01 deg; joints [29.046, -48.047, 113.734, -148.768, 69.512, 169.053] to (-171.06, -19.62, -54.5) mm, rotated rx 180 ry 0 rz 0.01 deg; joints [29.072, -48.157, 113.984, -148.768, 69.637, 169.121]
  MoveL 6131 to (-113.77, -19.62, -54.5) mm, rotated rx 180 ry 0 rz 0.01 deg; joints [30.266, -50.024, 118.218, -147.963, 71.898, 170.015]
  MoveC 6132 to (-112.41, -18.52, -54.5) mm, rotated rx 180 ry 0 rz 0.01 deg; joints [30.336, -50.048, 118.27, -147.895, 71.935, 170.008] to (-113.2, -16.96, -54.5) mm, rotated rx 180 ry 0 rz 0.01 deg; joints [30.377, -49.995, 118.147, -147.841, 71.884, 169.955]
  MoveL 6133 to (-186.65, 15.86, -54.5) mm, rotated rx -180 ry 0 rz 0.01 deg; joints [30.02, -46.986, 111.283, -147.47, 68.549, 167.892]
  MoveC 6134 to (-189.03, 17.2, -54.5) mm, rotated rx 180 ry 0 rz 0.01 deg; joints [30.019, -46.88, 111.042, -147.443, 68.436, 167.815] to (-191.14, 18.93, -54.5) mm, rotated rx -180 ry 0 rz 0.01 deg; joints [30.037, -46.775, 110.805, -147.396, 68.328, 167.732]
  MoveC 6135 to (-193.01, 20.91, -54.5) mm, rotated rx -180 ry 0 rz 0.01 deg; joints [30.068, -46.673, 110.575, -147.335, 68.227, 167.644] to (-194.74, 23.02, -54.5) mm, rotated rx 180 ry 0 rz 0.01 deg; joints [30.107, -46.574, 110.35, -147.268, 68.131, 167.556]
  MoveC 6136 to (-196.82, 24.04, -54.5) mm, rotated rx 180 ry 0 rz 0.01 deg; joints [30.1, -46.483, 110.145, -147.25, 68.034, 167.492] to (-198.86, 22.95, -54.5) mm, rotated rx 180 ry 0 rz 0.01 deg; joints [30.021, -46.433, 110.036, -147.32, 67.965, 167.49]
  MoveC 6137 to (-199.89, 21.56, -54.5) mm, rotated rx 180 ry 0 rz 0.01 deg; joints [29.952, -46.424, 110.019, -147.39, 67.942, 167.513] to (-200.99, 20.24, -54.5) mm, rotated rx -180 ry 0 rz 0.01 deg; joints [29.884, -46.41, 109.992, -147.458, 67.914, 167.532]
  MoveC 6138 to (-202.22, 19.03, -54.5) mm, rotated rx 180 ry 0 rz 0.01 deg; joints [29.818, -46.391, 109.952, -147.523, 67.88, 167.547] to (-203.59, 17.98, -54.5) mm, rotated rx 180 ry 0 rz 0.01 deg; joints [29.754, -46.363, 109.892, -147.583, 67.838, 167.554]
  MoveC 6139 to (-204.51, 17.36, -54.5) mm, rotated rx -180 ry 0 rz 0.01 deg; joints [29.714, -46.343, 109.848, -147.619, 67.809, 167.557] to (-205.41, 16.71, -54.5) mm, rotated rx 180 ry 0 rz 0.01 deg; joints [29.674, -46.324, 109.807, -147.657, 67.781, 167.561]
  MoveC 6140 to (-206.34, 16.1, -54.5) mm, rotated rx -180 ry 0 rz 0.01 deg; joints [29.634, -46.303, 109.762, -147.693, 67.751, 167.563] to (-207.32, 15.59, -54.5) mm, rotated rx 180 ry 0 rz 0.01 deg; joints [29.597, -46.278, 109.708, -147.726, 67.718, 167.561]
  MoveL 6141 to (-280.29, -16.96, -54.5) mm, rotated rx -180 ry 0 rz 0.01 deg; joints [27.11, -44.246, 105.294, -149.82, 65.08, 167.295]
  MoveC 6142 to (-281.08, -18.52, -54.5) mm, rotated rx 180 ry 0 rz 0.01 deg; joints [27.043, -44.245, 105.295, -149.893, 65.065, 167.327] to (-279.72, -19.62, -54.5) mm, rotated rx -180 ry 0 rz 0.01 deg; joints [27.029, -44.316, 105.452, -149.928, 65.137, 167.381]
  MoveL 6143 to (-171.06, -19.62, -54.5) mm, rotated rx 180 ry 0 rz 0.01 deg; joints [29.072, -48.157, 113.984, -148.768, 69.637, 169.121]
  MoveL 6144 to (-170.45, -19.47, -54.33) mm, rotated rx 180 ry 0 rz 0.01 deg; joints [29.09, -48.185, 114.025, -148.752, 69.652, 169.121]
  MoveL 6145 to (-170.09, -19.17, -53.87) mm, rotated rx 180 ry 0 rz 0.01 deg; joints [29.107, -48.219, 114.043, -148.73, 69.642, 169.106]
  MoveL 6146 to (-169.99, -19.04, -53.23) mm, rotated rx 180 ry 0 rz 0.01 deg; joints [29.114, -48.257, 114.049, -148.717, 69.616, 169.086]
  Set speed (500.0 mm/s)
  MoveL 6147 to (-169.99, -19.04, 11) mm, rotated rx -180 ry 0 rz 0.01 deg; joints [29.072, -51.926, 114.284, -148.039, 66.682, 167.163]
  Set speed (500.0 mm/s)
  MoveL 6148 to (-57.22, 262.99, 11) mm, rotated rx -180 ry 0 rz 0.01 deg; joints [41.038, -49.172, 108.111, -134.773, 67.679, 159.893]
  Set speed (500.0 mm/s)
  MoveL 6149 to (-57.22, 262.99, -32.73) mm, rotated rx 180 ry 0 rz 0.01 deg; joints [41.057, -46.846, 107.994, -135.369, 69.25, 161.563]
  Set speed (100.0 mm/s)
  MoveL 6150 to (-57.22, 263.15, -33.35) mm, rotated rx 180 ry 0 rz 0.01 deg; joints [41.062, -46.808, 107.982, -135.371, 69.27, 161.58]
  MoveL 6151 to (-57.23, 263.6, -33.82) mm, rotated rx -180 ry 0 rz 0.01 deg; joints [41.075, -46.771, 107.952, -135.36, 69.28, 161.581]
  MoveL 6152 to (-57.31, 264.21, -34) mm, rotated rx -180 ry 0 rz 0.01 deg; joints [41.091, -46.742, 107.91, -135.34, 69.276, 161.565]
  MoveL 6153 to (-61.83, 269.02, -34.24) mm, rotated rx 180 ry 0 rz 0.01 deg; joints [41.117, -46.456, 107.315, -135.231, 69.064, 161.322]
  MoveL 6154 to (-68.06, 266.8, -34.49) mm, rotated rx -180 ry 0 rz 0.01 deg; joints [40.891, -46.305, 107.019, -135.419, 68.885, 161.298]
  MoveL 6155 to (-68.52, 260.21, -34.73) mm, rotated rx -180 ry 0 rz 0.01 deg; joints [40.684, -46.453, 107.377, -135.684, 68.963, 161.532]
  MoveL 6156 to (-62.67, 257.15, -34.98) mm, rotated rx 180 ry 0 rz 0.01 deg; joints [40.743, -46.708, 107.957, -135.712, 69.216, 161.753]
  MoveL 6157 to (-57.52, 261.29, -35.22) mm, rotated rx -180 ry 0 rz 0.01 deg; joints [40.999, -46.748, 108.063, -135.471, 69.35, 161.709]
  MoveL 6158 to (-59.24, 267.66, -35.46) mm, rotated rx -180 ry 0 rz 0.01 deg; joints [41.144, -46.51, 107.567, -135.257, 69.215, 161.462]
  MoveL 6159 to (-65.77, 268.64, -35.71) mm, rotated rx -180 ry 0 rz 0.01 deg; joints [41.005, -46.263, 107.061, -135.328, 68.983, 161.319]
  MoveL 6160 to (-69.28, 263.04, -35.95) mm, rotated rx -180 ry 0 rz 0.01 deg; joints [40.749, -46.288, 107.151, -135.602, 68.942, 161.463]
  MoveL 6161 to (-65.56, 257.58, -36.2) mm, rotated rx 180 ry 0 rz 0.01 deg; joints [40.682, -46.538, 107.727, -135.757, 69.153, 161.731]
  MoveL 6162 to (-59.07, 258.8, -36.44) mm, rotated rx -180 ry 0 rz 0.01 deg; joints [40.886, -46.698, 108.098, -135.608, 69.371, 161.814]
  MoveL 6163 to (-57.59, 265.24, -36.68) mm, rotated rx -180 ry 0 rz 0.01 deg; joints [41.116, -46.561, 107.817, -135.339, 69.347, 161.623]
  MoveL 6164 to (-62.89, 269.18, -36.93) mm, rotated rx 180 ry 0 rz 0.01 deg; joints [41.095, -46.274, 107.221, -135.276, 69.119, 161.396]
  MoveL 6165 to (-68.62, 265.9, -37.17) mm, rotated rx 180 ry 0 rz 0.01 deg; joints [40.851, -46.167, 107.021, -135.497, 68.971, 161.418]
  MoveL 6166 to (-67.92, 259.33, -37.42) mm, rotated rx 180 ry 0 rz 0.01 deg; joints [40.675, -46.351, 107.457, -135.743, 69.09, 161.672]
  MoveL 6167 to (-61.62, 257.35, -37.66) mm, rotated rx -180 ry 0 rz 0.01 deg; joints [40.777, -46.591, 108.004, -135.721, 69.345, 161.864]
  MoveL 6168 to (-57.28, 262.32, -37.9) mm, rotated rx -180 ry 0 rz 0.01 deg; joints [41.038, -46.582, 108.005, -135.461, 69.439, 161.776]
  MoveL 6169 to (-60.09, 268.3, -38.15) mm, rotated rx 180 ry 0 rz 0.01 deg; joints [41.142, -46.321, 107.458, -135.281, 69.271, 161.523]
  MoveL 6170 to (-66.7, 268.11, -38.39) mm, rotated rx 180 ry 0 rz 0.01 deg; joints [40.967, -46.104, 107.016, -135.397, 69.052, 161.419]
  MoveL 6171 to (-69.17, 261.98, -38.64) mm, rotated rx -180 ry 0 rz 0.01 deg; joints [40.722, -46.176, 107.209, -135.676, 69.055, 161.6]
  MoveL 6172 to (-64.55, 257.26, -38.88) mm, rotated rx -180 ry 0 rz 0.01 deg; joints [40.7, -46.434, 107.803, -135.787, 69.287, 161.859]
  MoveL 6173 to (-58.37, 259.61, -39.12) mm, rotated rx 180 ry 0 rz 0.01 deg; joints [40.929, -46.554, 108.085, -135.599, 69.48, 161.897]
  MoveL 6174 to (-58.04, 266.2, -39.37) mm, rotated rx 180 ry 0 rz 0.01 deg; joints [41.134, -46.376, 107.716, -135.343, 69.413, 161.679]
  MoveL 6175 to (-63.96, 269.15, -39.61) mm, rotated rx -180 ry 0 rz 0.01 deg; joints [41.068, -46.097, 107.136, -135.329, 69.176, 161.476]
  MoveL 6176 to (-69.02, 264.91, -39.86) mm, rotated rx 180 ry 0 rz 0.01 deg; joints [40.813, -46.037, 107.039, -135.576, 69.064, 161.543]
  MoveL 6177 to (-67.17, 258.57, -40.1) mm, rotated rx 180 ry 0 rz 0.01 deg; joints [40.672, -46.25, 107.54, -135.794, 69.221, 161.81]
  MoveL 6178 to (-60.62, 257.73, -40.35) mm, rotated rx -180 ry 0 rz 0.01 deg; joints [40.815, -46.466, 108.037, -135.724, 69.47, 161.967]
  MoveL 6179 to (-57.22, 263.39, -40.59) mm, rotated rx 180 ry 0 rz 0.01 deg; joints [41.072, -46.41, 107.933, -135.453, 69.522, 161.838]
  MoveL 6180 to (-61.05, 268.77, -40.83) mm, rotated rx -180 ry 0 rz 0.01 deg; joints [41.133, -46.133, 107.351, -135.312, 69.325, 161.587]
  MoveL 6181 to (-67.51, 267.42, -41.08) mm, rotated rx -180 ry 0 rz 0.01 deg; joints [40.927, -45.952, 106.987, -135.47, 69.126, 161.526]
  MoveL 6182 to (-68.87, 260.96, -41.32) mm, rotated rx -180 ry 0 rz 0.01 deg; joints [40.7, -46.068, 107.276, -135.744, 69.173, 161.739]
  MoveL 6183 to (-63.49, 257.13, -41.57) mm, rotated rx 180 ry 0 rz 0.01 deg; joints [40.724, -46.326, 107.87, -135.808, 69.421, 161.98]
  MoveL 6184 to (-57.82, 260.52, -41.81) mm, rotated rx 180 ry 0 rz 0.01 deg; joints [40.972, -46.401, 108.055, -135.588, 69.582, 161.973]
  MoveL 6185 to (-58.66, 267.07, -42.05) mm, rotated rx 180 ry 0 rz 0.01 deg; joints [41.144, -46.188, 107.609, -135.353, 69.474, 161.735]
  MoveL 6186 to (-65, 268.93, -42.3) mm, rotated rx -180 ry 0 rz 0.01 deg; joints [41.036, -45.925, 107.064, -135.388, 69.236, 161.563]
  MoveL 6187 to (-69.24, 263.87, -42.54) mm, rotated rx 180 ry 0 rz 0.01 deg; joints [40.778, -45.913, 107.072, -135.653, 69.164, 161.674]
  MoveL 6188 to (-66.3, 257.95, -42.79) mm, rotated rx 180 ry 0 rz 0.01 deg; joints [40.677, -46.149, 107.622, -135.837, 69.355, 161.945]
  MoveL 6189 to (-59.71, 258.27, -43.03) mm, rotated rx 180 ry 0 rz 0.01 deg; joints [40.857, -46.335, 108.053, -135.721, 69.59, 162.062]
  MoveL 6190 to (-57.36, 264.45, -43.27) mm, rotated rx -180 ry 0 rz 0.01 deg; joints [41.101, -46.232, 107.847, -135.448, 69.597, 161.896]
  MoveL 6191 to (-62.07, 269.07, -43.52) mm, rotated rx -180 ry 0 rz 0.01 deg; joints [41.116, -45.948, 107.249, -135.35, 69.379, 161.656]
  MoveL 6192 to (-68.2, 266.61, -43.76) mm, rotated rx -180 ry 0 rz 0.01 deg; joints [40.886, -45.807, 106.975, -135.546, 69.206, 161.64]
  MoveL 6193 to (-68.39, 260, -44.01) mm, rotated rx 180 ry 0 rz 0.01 deg; joints [40.685, -45.963, 107.351, -135.807, 69.296, 161.879]
  MoveL 6194 to (-62.42, 257.18, -44.25) mm, rotated rx -180 ry 0 rz 0.01 deg; joints [40.754, -46.212, 107.925, -135.822, 69.552, 162.095]
  MoveL 6195 to (-57.44, 261.52, -44.49) mm, rotated rx 180 ry 0 rz 0.01 deg; joints [41.012, -46.24, 108.008, -135.577, 69.676, 162.042]
  MoveL 6196 to (-59.42, 267.82, -44.74) mm, rotated rx -180 ry 0 rz 0.01 deg; joints [41.148, -45.999, 107.498, -135.37, 69.531, 161.793]
  MoveL 6197 to (-65.99, 268.53, -44.98) mm, rotated rx -180 ry 0 rz 0.01 deg; joints [41, -45.76, 107.006, -135.452, 69.3, 161.656]
  MoveL 6198 to (-69.27, 262.8, -45.23) mm, rotated rx 180 ry 0 rz 0.01 deg; joints [40.747, -45.795, 107.119, -135.728, 69.271, 161.808]
  MoveL 6199 to (-65.34, 257.5, -45.47) mm, rotated rx 180 ry 0 rz 0.01 deg; joints [40.69, -46.046, 107.701, -135.872, 69.489, 162.075]
  MoveL 6200 to (-58.9, 258.98, -45.71) mm, rotated rx 180 ry 0 rz 0.01 deg; joints [40.899, -46.195, 108.052, -135.713, 69.703, 162.15]
  MoveL 6201 to (-57.68, 265.47, -45.96) mm, rotated rx -180 ry 0 rz 0.01 deg; joints [41.124, -46.049, 107.75, -135.447, 69.666, 161.952]
  MoveL 6202 to (-63.13, 269.19, -46.2) mm, rotated rx 180 ry 0 rz 0.01 deg; joints [41.093, -45.767, 107.155, -135.396, 69.433, 161.73]
  MoveL 6203 to (-68.73, 265.68, -46.45) mm, rotated rx 180 ry 0 rz 0.01 deg; joints [40.846, -45.67, 106.979, -135.624, 69.293, 161.76]
  MoveL 6204 to (-67.76, 259.15, -46.69) mm, rotated rx -180 ry 0 rz 0.01 deg; joints [40.677, -45.86, 107.43, -135.863, 69.424, 162.017]
  MoveL 6205 to (-61.38, 257.42, -46.93) mm, rotated rx -180 ry 0 rz 0.01 deg; joints [40.79, -46.092, 107.967, -135.829, 69.68, 162.203]
  MoveL 6206 to (-57.25, 262.57, -47.18) mm, rotated rx 180 ry 0 rz 0.01 deg; joints [41.05, -46.073, 107.944, -135.566, 69.763, 162.107]
  MoveL 6207 to (-60.3, 268.42, -47.42) mm, rotated rx -180 ry 0 rz 0.01 deg; joints [41.144, -45.81, 107.387, -135.395, 69.585, 161.853]
  MoveL 6208 to (-66.89, 267.96, -47.67) mm, rotated rx -180 ry 0 rz 0.01 deg; joints [40.961, -45.602, 106.962, -135.522, 69.369, 161.757]
  MoveL 6209 to (-69.12, 261.75, -47.91) mm, rotated rx 180 ry 0 rz 0.01 deg; joints [40.72, -45.683, 107.177, -135.799, 69.384, 161.945]
  MoveL 6210 to (-64.31, 257.22, -48.15) mm, rotated rx 180 ry 0 rz 0.01 deg; joints [40.709, -45.939, 107.772, -135.899, 69.623, 162.201]
  MoveL 6211 to (-58.23, 259.81, -48.4) mm, rotated rx 180 ry 0 rz 0.01 deg; joints [40.943, -46.048, 108.033, -135.703, 69.809, 162.23]
  MoveL 6212 to (-58.17, 266.41, -48.64) mm, rotated rx 180 ry 0 rz 0.01 deg; joints [41.14, -45.863, 107.645, -135.452, 69.73, 162.008]
  MoveL 6213 to (-64.2, 269.11, -48.89) mm, rotated rx -180 ry 0 rz 0.01 deg; joints [41.065, -45.59, 107.072, -135.449, 69.49, 161.81]
  MoveL 6214 to (-69.09, 264.68, -49.13) mm, rotated rx -180 ry 0 rz 0.01 deg; joints [40.809, -45.541, 106.998, -135.701, 69.387, 161.885]
  MoveL 6215 to (-66.98, 258.42, -49.38) mm, rotated rx 180 ry 0 rz 0.01 deg; joints [40.677, -45.758, 107.512, -135.911, 69.556, 162.154]
  MoveL 6216 to (-60.4, 257.84, -49.62) mm, rotated rx 180 ry 0 rz 0.01 deg; joints [40.828, -45.965, 107.994, -135.829, 69.803, 162.303]
  MoveL 6217 to (-57.24, 263.63, -49.86) mm, rotated rx 180 ry 0 rz 0.01 deg; joints [41.083, -45.899, 107.866, -135.558, 69.843, 162.167]
  MoveL 6218 to (-61.28, 268.86, -50.11) mm, rotated rx 180 ry 0 rz 0.01 deg; joints [41.133, -45.622, 107.279, -135.427, 69.638, 161.917]
  MoveL 6219 to (-67.68, 267.25, -50.35) mm, rotated rx -180 ry 0 rz 0.01 deg; joints [40.921, -45.451, 106.935, -135.595, 69.444, 161.864]
  MoveL 6220 to (-68.78, 260.73, -50.6) mm, rotated rx 180 ry 0 rz 0.01 deg; joints [40.7, -45.575, 107.245, -135.866, 69.503, 162.083]
  MoveL 6221 to (-63.25, 257.12, -50.84) mm, rotated rx -180 ry 0 rz 0.01 deg; joints [40.735, -45.829, 107.835, -135.918, 69.756, 162.32]
  MoveL 6222 to (-57.72, 260.74, -51.08) mm, rotated rx -180 ry 0 rz 0.01 deg; joints [40.985, -45.893, 107.997, -135.691, 69.908, 162.303]
  MoveL 6223 to (-58.82, 267.25, -51.33) mm, rotated rx 180 ry 0 rz 0.01 deg; joints [41.15, -45.674, 107.535, -135.463, 69.788, 162.063]
  MoveL 6224 to (-65.23, 268.85, -51.57) mm, rotated rx -180 ry 0 rz 0.01 deg; joints [41.032, -45.419, 107.001, -135.509, 69.55, 161.896]
  MoveL 6225 to (-69.26, 263.62, -51.82) mm, rotated rx 180 ry 0 rz 0.01 deg; joints [40.774, -45.417, 107.033, -135.777, 69.489, 162.016]
  MoveL 6226 to (-66.09, 257.83, -52.06) mm, rotated rx 180 ry 0 rz 0.01 deg; joints [40.683, -45.655, 107.591, -135.952, 69.689, 162.287]
  MoveL 6227 to (-59.51, 258.42, -52.3) mm, rotated rx 180 ry 0 rz 0.01 deg; joints [40.87, -45.831, 108.005, -135.824, 69.921, 162.396]
  MoveL 6228 to (-57.41, 264.68, -52.55) mm, rotated rx -180 ry 0 rz 0.01 deg; joints [41.111, -45.719, 107.776, -135.552, 69.916, 162.223]
  MoveL 6229 to (-62.31, 269.12, -52.79) mm, rotated rx -180 ry 0 rz 0.01 deg; joints [41.115, -45.437, 107.177, -135.466, 69.691, 161.985]
  MoveL 6230 to (-68.33, 266.4, -53.04) mm, rotated rx 180 ry 0 rz 0.01 deg; joints [40.881, -45.307, 106.925, -135.67, 69.525, 161.978]
  MoveL 6231 to (-68.26, 259.8, -53.28) mm, rotated rx 180 ry 0 rz 0.01 deg; joints [40.687, -45.469, 107.319, -135.926, 69.628, 162.221]
  MoveL 6232 to (-62.18, 257.22, -53.52) mm, rotated rx 180 ry 0 rz 0.01 deg; joints [40.766, -45.713, 107.886, -135.929, 69.886, 162.433]
  MoveL 6233 to (-57.38, 261.75, -53.77) mm, rotated rx -180 ry 0 rz 0.01 deg; joints [41.025, -45.73, 107.944, -135.679, 70, 162.371]
  MoveL 6234 to (-59.62, 267.97, -54.01) mm, rotated rx 180 ry 0 rz 0.01 deg; joints [41.152, -45.485, 107.422, -135.481, 69.844, 162.119]
  MoveL 6235 to (-66.2, 268.42, -54.26) mm, rotated rx -180 ry 0 rz 0.01 deg; joints [40.995, -45.255, 106.944, -135.574, 69.615, 161.99]
  MoveL 6236 to (-69.25, 262.56, -54.5) mm, rotated rx 180 ry 0 rz 0.01 deg; joints [40.744, -45.3, 107.08, -135.85, 69.597, 162.149]
  MoveL 6237 to (-65.15, 221.39, -54.5) mm, rotated rx 180 ry 0 rz 0.01 deg; joints [39.604, -46.475, 109.744, -137.374, 70.318, 163.644]
  MoveC 6238 to (-63.95, 220.36, -54.5) mm, rotated rx -180 ry 0 rz 0.01 deg; joints [39.603, -46.538, 109.885, -137.394, 70.375, 163.701] to (-62.86, 221.5, -54.5) mm, rotated rx 180 ry 0 rz 0.01 deg; joints [39.666, -46.543, 109.894, -137.331, 70.397, 163.682]
  MoveL 6239 to (-62.86, 263.24, -54.5) mm, rotated rx 180 ry 0 rz 0.01 deg; joints [40.928, -45.481, 107.478, -135.721, 69.813, 162.244]
  MoveC 6240 to (-63.69, 265.25, -54.5) mm, rotated rx -180 ry 0 rz 0.01 deg; joints [40.966, -45.403, 107.302, -135.657, 69.756, 162.158] to (-65.7, 266.08, -54.5) mm, rotated rx -180 ry 0 rz 0.01 deg; joints [40.939, -45.319, 107.116, -135.658, 69.673, 162.091]
  MoveL 6241 to (-66.47, 266.08, -54.5) mm, rotated rx 180 ry 0 rz 0.01 deg; joints [40.919, -45.295, 107.063, -135.67, 69.646, 162.077]
  MoveC 6242 to (-68.57, 265.15, -54.5) mm, rotated rx 180 ry 0 rz 0.01 deg; joints [40.838, -45.253, 106.974, -135.74, 69.585, 162.07] to (-69.29, 262.96, -54.5) mm, rotated rx -180 ry 0 rz 0.01 deg; joints [40.755, -45.288, 107.054, -135.836, 69.59, 162.134]
  MoveL 6243 to (-69.25, 262.56, -54.5) mm, rotated rx 180 ry 0 rz 0.01 deg; joints [40.744, -45.3, 107.08, -135.85, 69.597, 162.149]
  MoveC 6244 to (-69.73, 260.11, -54.5) mm, rotated rx -180 ry 0 rz 0.01 deg; joints [40.659, -45.349, 107.192, -135.952, 69.614, 162.226] to (-71.49, 258.34, -54.5) mm, rotated rx 180 ry 0 rz 0.01 deg; joints [40.562, -45.34, 107.175, -136.048, 69.577, 162.256]
  MoveC 6245 to (-73.25, 256.58, -54.5) mm, rotated rx -180 ry 0 rz 0.01 deg; joints [40.464, -45.331, 107.158, -136.144, 69.539, 162.285] to (-73.73, 254.13, -54.5) mm, rotated rx -180 ry 0 rz 0.01 deg; joints [40.379, -45.379, 107.268, -136.246, 69.556, 162.362]
  MoveL 6246 to (-66.93, 185.98, -54.5) mm, rotated rx -180 ry 0 rz 0.01 deg; joints [38.452, -47.276, 111.588, -138.788, 70.754, 164.785]
  MoveC 6247 to (-66.44, 184.46, -54.5) mm, rotated rx 180 ry 0 rz 0.01 deg; joints [38.416, -47.327, 111.705, -138.839, 70.793, 164.843] to (-65.37, 183.27, -54.5) mm, rotated rx 180 ry 0 rz 0.01 deg; joints [38.405, -47.389, 111.843, -138.868, 70.848, 164.9]
  MoveL 6248 to (-60.81, 179.99, -54.5) mm, rotated rx -180 ry 0 rz 0.01 deg; joints [38.416, -47.605, 112.333, -138.919, 71.057, 165.087]
  MoveC 6249 to (-58.68, 179.83, -54.5) mm, rotated rx -180 ry 0 rz 0.01 deg; joints [38.465, -47.674, 112.487, -138.889, 71.135, 165.129] to (-57.57, 181.66, -54.5) mm, rotated rx -180 ry 0 rz 0.01 deg; joints [38.552, -47.666, 112.464, -138.798, 71.148, 165.09]
  MoveL 6250 to (-57.57, 267.52, -54.5) mm, rotated rx -180 ry 0 rz 0.01 deg; joints [41.191, -45.533, 107.585, -135.47, 69.939, 162.191]
  MoveC 6251 to (-58.7, 270.24, -54.5) mm, rotated rx 180 ry 0 rz 0.01 deg; joints [41.243, -45.427, 107.346, -135.384, 69.861, 162.074] to (-61.42, 271.37, -54.5) mm, rotated rx 180 ry 0 rz 0.01 deg; joints [41.205, -45.312, 107.093, -135.386, 69.75, 161.983]
  MoveL 6252 to (-71.67, 271.37, -54.5) mm, rotated rx 180 ry 0 rz 0.01 deg; joints [40.943, -44.992, 106.39, -135.55, 69.389, 161.792]
  MoveC 6253 to (-74.21, 270.24, -54.5) mm, rotated rx 180 ry 0 rz 0.01 deg; joints [40.845, -44.942, 106.282, -135.634, 69.315, 161.784] to (-75.08, 267.61, -54.5) mm, rotated rx -180 ry 0 rz 0.01 deg; joints [40.745, -44.985, 106.379, -135.749, 69.321, 161.862]
  MoveL 6254 to (-73.73, 254.13, -54.5) mm, rotated rx 180 ry 0 rz 0.01 deg; joints [40.379, -45.379, 107.268, -136.246, 69.556, 162.362]
  MoveC 6255 to (-74.44, 250.52, -54.5) mm, rotated rx -180 ry 0 rz 0.01 deg; joints [40.253, -45.45, 107.43, -136.397, 69.581, 162.475] to (-77.04, 247.92, -54.5) mm, rotated rx -180 ry 0 rz 0.01 deg; joints [40.109, -45.435, 107.403, -136.539, 69.525, 162.518]
  MoveC 6256 to (-79.63, 245.31, -54.5) mm, rotated rx -180 ry 0 rz 0.01 deg; joints [39.965, -45.42, 107.374, -136.681, 69.469, 162.56] to (-80.34, 241.7, -54.5) mm, rotated rx -180 ry 0 rz 0.01 deg; joints [39.839, -45.49, 107.534, -136.832, 69.494, 162.672]
  MoveL 6257 to (-74.73, 185.45, -54.5) mm, rotated rx -180 ry 0 rz 0.01 deg; joints [38.239, -47.048, 111.08, -138.939, 70.482, 164.664]
  MoveC 6258 to (-73.16, 180.58, -54.5) mm, rotated rx 180 ry 0 rz 0.01 deg; joints [38.124, -47.211, 111.452, -139.105, 70.607, 164.85] to (-69.73, 176.78, -54.5) mm, rotated rx -180 ry 0 rz 0.01 deg; joints [38.089, -47.406, 111.894, -139.197, 70.784, 165.033]
  MoveL 6259 to (-53, 164.76, -54.5) mm, rotated rx -180 ry 0 rz 0.01 deg; joints [38.124, -48.196, 113.684, -139.384, 71.551, 165.71]
  MoveC 6260 to (-50.87, 164.6, -54.5) mm, rotated rx -180 ry 0 rz 0.01 deg; joints [38.173, -48.264, 113.837, -139.352, 71.629, 165.752] to (-49.76, 166.43, -54.5) mm, rotated rx -180 ry 0 rz 0.01 deg; joints [38.261, -48.256, 113.815, -139.26, 71.642, 165.714]
  MoveL 6261 to (-49.76, 275.33, -54.5) mm, rotated rx -180 ry 0 rz 0.01 deg; joints [41.625, -45.568, 107.648, -135.042, 70.102, 162.059]
  MoveC 6262 to (-50.89, 278.05, -54.5) mm, rotated rx 180 ry 0 rz 0.01 deg; joints [41.675, -45.461, 107.409, -134.957, 70.025, 161.941] to (-53.61, 279.18, -54.5) mm, rotated rx -180 ry 0 rz 0.01 deg; joints [41.637, -45.347, 107.156, -134.96, 69.914, 161.85]
  MoveL 6263 to (-80.3, 279.18, -54.5) mm, rotated rx -180 ry 0 rz 0.01 deg; joints [40.952, -44.512, 105.325, -135.385, 68.976, 161.349]
  MoveC 6264 to (-82.83, 278.05, -54.5) mm, rotated rx 180 ry 0 rz 0.01 deg; joints [40.855, -44.462, 105.216, -135.467, 68.901, 161.342] to (-83.7, 275.42, -54.5) mm, rotated rx -180 ry 0 rz 0.01 deg; joints [40.756, -44.504, 105.314, -135.581, 68.906, 161.42]
  MoveL 6265 to (-80.34, 241.7, -54.5) mm, rotated rx -180 ry 0 rz 0.01 deg; joints [39.839, -45.49, 107.534, -136.832, 69.494, 162.672]
  MoveC 6266 to (-81.05, 238.09, -54.5) mm, rotated rx 180 ry 0 rz 0.01 deg; joints [39.712, -45.56, 107.693, -136.983, 69.518, 162.784] to (-83.64, 235.48, -54.5) mm, rotated rx 180 ry 0 rz 0.01 deg; joints [39.568, -45.544, 107.663, -137.125, 69.462, 162.826]
  MoveC 6267 to (-86.24, 232.88, -54.5) mm, rotated rx 180 ry 0 rz 0.01 deg; joints [39.424, -45.528, 107.632, -137.267, 69.405, 162.868] to (-86.95, 229.27, -54.5) mm, rotated rx 180 ry 0 rz 0.01 deg; joints [39.296, -45.596, 107.788, -137.419, 69.43, 162.979]
  MoveL 6268 to (-82.18, 181.49, -54.5) mm, rotated rx -180 ry 0 rz 0.01 deg; joints [37.928, -46.908, 110.777, -139.217, 70.269, 164.66]
  MoveC 6269 to (-80.52, 176.33, -54.5) mm, rotated rx -180 ry 0 rz 0.01 deg; joints [37.805, -47.081, 111.172, -139.394, 70.402, 164.857] to (-76.88, 172.31, -54.5) mm, rotated rx 180 ry 0 rz 0.01 deg; joints [37.767, -47.288, 111.64, -139.494, 70.59, 165.051]
  MoveL 6270 to (-45.19, 149.53, -54.5) mm, rotated rx -180 ry 0 rz 0.01 deg; joints [37.825, -48.776, 115.018, -139.848, 72.047, 166.322]
  MoveC 6271 to (-43.06, 149.37, -54.5) mm, rotated rx 180 ry 0 rz 0.01 deg; joints [37.875, -48.844, 115.171, -139.815, 72.125, 166.364] to (-41.95, 151.2, -54.5) mm, rotated rx -180 ry 0 rz 0.01 deg; joints [37.963, -48.836, 115.15, -139.723, 72.138, 166.327]
  MoveL 6272 to (-41.95, 283.14, -54.5) mm, rotated rx 180 ry 0 rz 0.01 deg; joints [42.058, -45.599, 107.704, -134.614, 70.263, 161.925]
  MoveC 6273 to (-43.08, 285.86, -54.5) mm, rotated rx -180 ry 0 rz 0.01 deg; joints [42.108, -45.492, 107.464, -134.53, 70.186, 161.807] to (-45.8, 286.99, -54.5) mm, rotated rx 180 ry 0 rz 0.01 deg; joints [42.069, -45.378, 107.212, -134.533, 70.076, 161.716]
  MoveL 6274 to (-88.92, 286.99, -54.5) mm, rotated rx 180 ry 0 rz 0.01 deg; joints [40.961, -44.026, 104.251, -135.215, 68.56, 160.902]
  MoveC 6275 to (-91.46, 285.86, -54.5) mm, rotated rx 180 ry 0 rz 0.01 deg; joints [40.865, -43.975, 104.141, -135.295, 68.485, 160.894] to (-92.33, 283.23, -54.5) mm, rotated rx 180 ry 0 rz 0.01 deg; joints [40.767, -44.019, 104.24, -135.41, 68.49, 160.973]
  MoveL 6276 to (-86.95, 229.27, -54.5) mm, rotated rx -180 ry 0 rz 0.01 deg; joints [39.296, -45.596, 107.788, -137.419, 69.43, 162.979]
  MoveC 6277 to (-87.66, 225.66, -54.5) mm, rotated rx -180 ry 0 rz 0.01 deg; joints [39.169, -45.664, 107.944, -137.57, 69.454, 163.089] to (-90.25, 223.05, -54.5) mm, rotated rx -180 ry 0 rz 0.01 deg; joints [39.024, -45.647, 107.911, -137.713, 69.397, 163.13]
  MoveC 6278 to (-92.84, 220.44, -54.5) mm, rotated rx 180 ry 0 rz 0.01 deg; joints [38.88, -45.629, 107.876, -137.855, 69.34, 163.171] to (-93.56, 216.84, -54.5) mm, rotated rx 180 ry 0 rz 0.01 deg; joints [38.752, -45.696, 108.03, -138.007, 69.364, 163.281]
  MoveL 6279 to (-89.6, 177.2, -54.5) mm, rotated rx 180 ry 0 rz 0.01 deg; joints [37.609, -46.775, 110.49, -139.506, 70.061, 164.667]
  MoveC 6280 to (-87.94, 172.04, -54.5) mm, rotated rx 180 ry 0 rz 0.01 deg; joints [37.485, -46.948, 110.884, -139.684, 70.193, 164.863] to (-84.3, 168.03, -54.5) mm, rotated rx 180 ry 0 rz 0.01 deg; joints [37.446, -47.156, 111.353, -139.785, 70.382, 165.057]
  MoveL 6281 to (-37.38, 134.3, -54.5) mm, rotated rx -180 ry 0 rz 0.01 deg; joints [37.52, -49.347, 116.338, -140.311, 72.544, 166.925]
  MoveC 6282 to (-35.25, 134.15, -54.5) mm, rotated rx 180 ry 0 rz 0.01 deg; joints [37.569, -49.413, 116.49, -140.278, 72.621, 166.966] to (-34.14, 135.97, -54.5) mm, rotated rx -180 ry 0 rz 0.01 deg; joints [37.659, -49.406, 116.47, -140.184, 72.634, 166.929]
  MoveL 6283 to (-34.14, 290.95, -54.5) mm, rotated rx -180 ry 0 rz 0.01 deg; joints [42.492, -45.627, 107.752, -134.184, 70.422, 161.79]
  MoveC 6284 to (-35.27, 293.67, -54.5) mm, rotated rx 180 ry 0 rz 0.01 deg; joints [42.541, -45.519, 107.511, -134.101, 70.346, 161.671] to (-37.99, 294.8, -54.5) mm, rotated rx 180 ry 0 rz 0.01 deg; joints [42.502, -45.406, 107.26, -134.105, 70.237, 161.58]
  MoveL 6285 to (-97.55, 294.8, -54.5) mm, rotated rx 180 ry 0 rz 0.01 deg; joints [40.971, -43.535, 103.167, -135.039, 68.144, 160.448]
  MoveC 6286 to (-100.09, 293.67, -54.5) mm, rotated rx 180 ry 0 rz 0.01 deg; joints [40.875, -43.483, 103.056, -135.119, 68.068, 160.44] to (-100.96, 291.04, -54.5) mm, rotated rx 180 ry 0 rz 0.01 deg; joints [40.777, -43.527, 103.156, -135.233, 68.073, 160.521]
  MoveL 6287 to (-93.56, 216.84, -54.5) mm, rotated rx -180 ry 0 rz 0.01 deg; joints [38.752, -45.696, 108.03, -138.007, 69.364, 163.281]
  MoveC 6288 to (-94.27, 213.22, -54.5) mm, rotated rx -180 ry 0 rz 0.01 deg; joints [38.623, -45.762, 108.183, -138.159, 69.389, 163.39] to (-96.86, 210.61, -54.5) mm, rotated rx -180 ry 0 rz 0.01 deg; joints [38.479, -45.744, 108.147, -138.302, 69.331, 163.431]
  MoveC 6289 to (-99.46, 208, -54.5) mm, rotated rx -180 ry 0 rz 0.01 deg; joints [38.334, -45.725, 108.109, -138.444, 69.273, 163.471] to (-100.17, 204.38, -54.5) mm, rotated rx -180 ry 0 rz 0.01 deg; joints [38.205, -45.79, 108.26, -138.597, 69.297, 163.58]
  MoveL 6290 to (-97.02, 172.92, -54.5) mm, rotated rx -180 ry 0 rz 0.01 deg; joints [37.291, -46.641, 110.199, -139.793, 69.85, 164.674]
  MoveC 6291 to (-95.36, 167.76, -54.5) mm, rotated rx -180 ry 0 rz 0.01 deg; joints [37.167, -46.813, 110.592, -139.972, 69.983, 164.87] to (-91.72, 163.74, -54.5) mm, rotated rx 180 ry 0 rz 0.01 deg; joints [37.126, -47.021, 111.061, -140.074, 70.172, 165.063]
  MoveL 6292 to (-29.57, 119.07, -54.5) mm, rotated rx 180 ry 0 rz 0.01 deg; joints [37.207, -49.907, 117.643, -140.775, 73.042, 167.517]
  MoveC 6293 to (-27.44, 118.92, -54.5) mm, rotated rx -180 ry 0 rz 0.01 deg; joints [37.257, -49.973, 117.794, -140.741, 73.12, 167.558] to (-26.33, 120.74, -54.5) mm, rotated rx -180 ry 0 rz 0.01 deg; joints [37.348, -49.967, 117.776, -140.646, 73.132, 167.522]
  MoveL 6294 to (-26.33, 298.76, -54.5) mm, rotated rx 180 ry 0 rz 0.01 deg; joints [42.927, -45.651, 107.793, -133.755, 70.58, 161.653]
  MoveC 6295 to (-27.46, 301.48, -54.5) mm, rotated rx 180 ry 0 rz 0.01 deg; joints [42.975, -45.543, 107.551, -133.672, 70.504, 161.534] to (-30.18, 302.61, -54.5) mm, rotated rx -180 ry 0 rz 0.01 deg; joints [42.934, -45.43, 107.301, -133.677, 70.395, 161.442]
  MoveL 6296 to (-106.25, 302.61, -54.5) mm, rotated rx 180 ry 0 rz 0.01 deg; joints [40.978, -43.035, 102.068, -134.86, 67.723, 159.988]
  MoveC 6297 to (-108.77, 301.48, -54.5) mm, rotated rx 180 ry 0 rz 0.01 deg; joints [40.883, -42.983, 101.957, -134.938, 67.647, 159.98] to (-109.62, 298.85, -54.5) mm, rotated rx 180 ry 0 rz 0.01 deg; joints [40.787, -43.028, 102.059, -135.051, 67.652, 160.061]
  MoveL 6298 to (-100.17, 204.38, -54.5) mm, rotated rx 180 ry 0 rz 0.01 deg; joints [38.205, -45.79, 108.26, -138.597, 69.297, 163.58]
  MoveC 6299 to (-100.88, 200.83, -54.5) mm, rotated rx -180 ry 0 rz 0.01 deg; joints [38.077, -45.854, 108.407, -138.748, 69.321, 163.686] to (-103.44, 198.27, -54.5) mm, rotated rx 180 ry 0 rz 0.01 deg; joints [37.935, -45.834, 108.367, -138.888, 69.263, 163.725]
  MoveC 6300 to (-106, 195.71, -54.5) mm, rotated rx 180 ry 0 rz 0.01 deg; joints [37.793, -45.813, 108.327, -139.028, 69.205, 163.764] to (-106.71, 192.16, -54.5) mm, rotated rx -180 ry 0 rz 0.01 deg; joints [37.665, -45.876, 108.471, -139.179, 69.228, 163.869]
  MoveL 6301 to (-104.35, 167.74, -54.5) mm, rotated rx -180 ry 0 rz 0.01 deg; joints [36.948, -46.527, 109.957, -140.112, 69.653, 164.71]
  MoveC 6302 to (-102.95, 163.38, -54.5) mm, rotated rx -180 ry 0 rz 0.01 deg; joints [36.842, -46.673, 110.288, -140.265, 69.766, 164.876] to (-99.88, 159.98, -54.5) mm, rotated rx -180 ry 0 rz 0.01 deg; joints [36.807, -46.849, 110.686, -140.353, 69.926, 165.039]
  MoveL 6303 to (-21.76, 103.84, -54.5) mm, rotated rx 180 ry 0 rz 0.01 deg; joints [36.887, -50.458, 118.934, -141.239, 73.542, 168.1]
  MoveC 6304 to (-19.63, 103.69, -54.5) mm, rotated rx -180 ry 0 rz 0.01 deg; joints [36.937, -50.524, 119.084, -141.204, 73.619, 168.14] to (-18.52, 105.51, -54.5) mm, rotated rx 180 ry 0 rz 0.01 deg; joints [37.029, -50.518, 119.067, -141.109, 73.632, 168.106]
  MoveL 6305 to (-18.52, 306.57, -54.5) mm, rotated rx 180 ry 0 rz 0.01 deg; joints [43.361, -45.671, 107.826, -133.324, 70.736, 161.514]
  MoveC 6306 to (-19.65, 309.29, -54.5) mm, rotated rx 180 ry 0 rz 0.01 deg; joints [43.409, -45.563, 107.583, -133.243, 70.66, 161.394] to (-22.37, 310.42, -54.5) mm, rotated rx -180 ry 0 rz 0.01 deg; joints [43.367, -45.451, 107.334, -133.249, 70.552, 161.303]
  MoveL 6307 to (-115.49, 310.42, -54.5) mm, rotated rx 180 ry 0 rz 0.01 deg; joints [40.972, -42.512, 100.92, -134.683, 67.281, 159.511]
  MoveC 6308 to (-117.83, 309.31, -54.5) mm, rotated rx 180 ry 0 rz 0.01 deg; joints [40.883, -42.465, 100.82, -134.756, 67.211, 159.505] to (-118.46, 306.79, -54.5) mm, rotated rx -180 ry 0 rz 0.01 deg; joints [40.796, -42.514, 100.931, -134.862, 67.222, 159.588]
  MoveC 6309 to (-117.28, 299.98, -54.5) mm, rotated rx 180 ry 0 rz 0.01 deg; joints [40.631, -42.744, 101.44, -135.111, 67.358, 159.867] to (-116.43, 293.11, -54.5) mm, rotated rx -180 ry 0 rz 0.01 deg; joints [40.456, -42.962, 101.923, -135.366, 67.483, 160.14]
  MoveL 6310 to (-106.71, 192.16, -54.5) mm, rotated rx -180 ry 0 rz 0.01 deg; joints [37.665, -45.876, 108.471, -139.179, 69.228, 163.869]
  MoveC 6311 to (-107.42, 188.6, -54.5) mm, rotated rx 180 ry 0 rz 0.01 deg; joints [37.536, -45.938, 108.615, -139.33, 69.251, 163.973] to (-109.98, 186.04, -54.5) mm, rotated rx -180 ry 0 rz 0.01 deg; joints [37.394, -45.916, 108.572, -139.47, 69.192, 164.012]
  MoveC 6312 to (-112.55, 183.48, -54.5) mm, rotated rx 180 ry 0 rz 0.01 deg; joints [37.252, -45.894, 108.528, -139.61, 69.133, 164.05] to (-113.26, 179.93, -54.5) mm, rotated rx 180 ry 0 rz 0.01 deg; joints [37.122, -45.955, 108.669, -139.762, 69.156, 164.153]
  MoveL 6313 to (-111.9, 165.83, -54.5) mm, rotated rx 180 ry 0 rz 0.01 deg; joints [36.707, -46.329, 109.522, -140.303, 69.401, 164.637]
  MoveC 6314 to (-111.84, 164.93, -54.5) mm, rotated rx 180 ry 0 rz 0.01 deg; joints [36.679, -46.352, 109.574, -140.338, 69.416, 164.667] to (-111.84, 164.03, -54.5) mm, rotated rx 180 ry 0 rz 0.01 deg; joints [36.65, -46.372, 109.621, -140.374, 69.428, 164.696]
  MoveC 6315 to (-111.88, 163.13, -54.5) mm, rotated rx 180 ry 0 rz 0.01 deg; joints [36.621, -46.392, 109.667, -140.411, 69.44, 164.725] to (-111.92, 162.23, -54.5) mm, rotated rx 180 ry 0 rz 0.01 deg; joints [36.591, -46.412, 109.711, -140.447, 69.451, 164.753]
  MoveC 6316 to (-111.05, 158.67, -54.5) mm, rotated rx 180 ry 0 rz 0.01 deg; joints [36.497, -46.521, 109.961, -140.577, 69.532, 164.883] to (-108.39, 156.14, -54.5) mm, rotated rx 180 ry 0 rz 0.01 deg; joints [36.479, -46.664, 110.284, -140.637, 69.665, 165.011]
  MoveC 6317 to (-107.58, 155.72, -54.5) mm, rotated rx 180 ry 0 rz 0.01 deg; joints [36.485, -46.7, 110.364, -140.641, 69.702, 165.039] to (-106.76, 155.3, -54.5) mm, rotated rx 180 ry 0 rz 0.01 deg; joints [36.491, -46.736, 110.445, -140.646, 69.738, 165.067]
  MoveC 6318 to (-105.96, 154.84, -54.5) mm, rotated rx 180 ry 0 rz 0.01 deg; joints [36.495, -46.772, 110.526, -140.652, 69.774, 165.096] to (-105.19, 154.32, -54.5) mm, rotated rx 180 ry 0 rz 0.01 deg; joints [36.497, -46.809, 110.607, -140.661, 69.809, 165.126]
  MoveL 6319 to (-13.95, 88.62, -54.5) mm, rotated rx -180 ry 0 rz 0.01 deg; joints [36.56, -51, 120.211, -141.704, 74.044, 168.673]
  MoveC 6320 to (-11.82, 88.46, -54.5) mm, rotated rx -180 ry 0 rz 0.01 deg; joints [36.61, -51.064, 120.36, -141.669, 74.121, 168.713] to (-10.7, 90.28, -54.5) mm, rotated rx 180 ry 0 rz 0.01 deg; joints [36.703, -51.059, 120.344, -141.573, 74.133, 168.68]
  MoveL 6321 to (-10.71, 314.38, -54.5) mm, rotated rx 180 ry 0 rz 0.01 deg; joints [43.796, -45.688, 107.851, -132.894, 70.889, 161.374]
  MoveC 6322 to (-11.84, 317.1, -54.5) mm, rotated rx -180 ry 0 rz 0.01 deg; joints [43.843, -45.58, 107.607, -132.813, 70.814, 161.253] to (-14.56, 318.23, -54.5) mm, rotated rx 180 ry 0 rz 0.01 deg; joints [43.8, -45.468, 107.359, -132.82, 70.706, 161.162]
  MoveL 6323 to (-125.78, 318.23, -54.5) mm, rotated rx -180 ry 0 rz 0.01 deg; joints [40.94, -41.946, 99.683, -134.512, 66.798, 159.005]
  MoveC 6324 to (-127.94, 317.15, -54.5) mm, rotated rx 180 ry 0 rz 0.01 deg; joints [40.857, -41.903, 99.593, -134.581, 66.734, 159.002] to (-128.39, 314.78, -54.5) mm, rotated rx 180 ry 0 rz 0.01 deg; joints [40.78, -41.956, 99.711, -134.679, 66.749, 159.083]
  MoveC 6325 to (-125.77, 303.74, -54.5) mm, rotated rx 180 ry 0 rz 0.01 deg; joints [40.531, -42.355, 100.591, -135.075, 66.996, 159.555] to (-124.11, 292.53, -54.5) mm, rotated rx 180 ry 0 rz 0.01 deg; joints [40.252, -42.722, 101.404, -135.49, 67.21, 160.009]
  MoveL 6326 to (-113.26, 179.93, -54.5) mm, rotated rx 180 ry 0 rz 0.01 deg; joints [37.122, -45.955, 108.669, -139.762, 69.156, 164.153]
  MoveC 6327 to (-113.96, 176.4, -54.5) mm, rotated rx -180 ry 0 rz 0.01 deg; joints [36.994, -46.016, 108.809, -139.912, 69.179, 164.256] to (-116.51, 173.86, -54.5) mm, rotated rx -180 ry 0 rz 0.01 deg; joints [36.853, -45.993, 108.764, -140.051, 69.12, 164.294]
  MoveC 6328 to (-119.05, 171.31, -54.5) mm, rotated rx -180 ry 0 rz 0.01 deg; joints [36.711, -45.97, 108.717, -140.19, 69.06, 164.331] to (-119.75, 167.78, -54.5) mm, rotated rx 180 ry 0 rz 0.01 deg; joints [36.582, -46.029, 108.855, -140.341, 69.083, 164.433]
  MoveL 6329 to (-119.49, 165.07, -54.5) mm, rotated rx 180 ry 0 rz 0.01 deg; joints [36.502, -46.101, 109.018, -140.446, 69.13, 164.526]
  MoveC 6330 to (-119.43, 162.68, -54.5) mm, rotated rx 180 ry 0 rz 0.01 deg; joints [36.427, -46.158, 109.149, -140.541, 69.166, 164.604] to (-119.72, 160.31, -54.5) mm, rotated rx -180 ry 0 rz 0.01 deg; joints [36.344, -46.203, 109.254, -140.64, 69.188, 164.676]
  MoveC 6331 to (-120.24, 157.98, -54.5) mm, rotated rx 180 ry 0 rz 0.01 deg; joints [36.257, -46.24, 109.339, -140.741, 69.2, 164.741] to (-120.9, 155.69, -54.5) mm, rotated rx -180 ry 0 rz 0.01 deg; joints [36.168, -46.271, 109.412, -140.842, 69.207, 164.803]
  MoveC 6332 to (-120.64, 153.19, -54.5) mm, rotated rx -180 ry 0 rz 0.01 deg; joints [36.094, -46.336, 109.562, -140.939, 69.251, 164.888] to (-118.63, 151.69, -54.5) mm, rotated rx 180 ry 0 rz 0.01 deg; joints [36.093, -46.436, 109.785, -140.969, 69.347, 164.971]
  MoveC 6333 to (-116.93, 151.26, -54.5) mm, rotated rx -180 ry 0 rz 0.01 deg; joints [36.119, -46.501, 109.93, -140.961, 69.417, 165.015] to (-115.24, 150.76, -54.5) mm, rotated rx -180 ry 0 rz 0.01 deg; joints [36.143, -46.567, 110.077, -140.956, 69.486, 165.061]
  MoveC 6334 to (-113.58, 150.17, -54.5) mm, rotated rx -180 ry 0 rz 0.01 deg; joints [36.163, -46.634, 110.226, -140.955, 69.556, 165.109] to (-111.97, 149.45, -54.5) mm, rotated rx 180 ry 0 rz 0.01 deg; joints [36.177, -46.702, 110.379, -140.96, 69.626, 165.161]
  MoveC 6335 to (-111.37, 149.14, -54.5) mm, rotated rx -180 ry 0 rz 0.01 deg; joints [36.182, -46.728, 110.438, -140.963, 69.652, 165.181] to (-110.78, 148.84, -54.5) mm, rotated rx 180 ry 0 rz 0.01 deg; joints [36.186, -46.754, 110.496, -140.966, 69.679, 165.201]
  MoveC 6336 to (-110.2, 148.51, -54.5) mm, rotated rx -180 ry 0 rz 0.01 deg; joints [36.189, -46.78, 110.555, -140.97, 69.705, 165.222] to (-109.64, 148.13, -54.5) mm, rotated rx 180 ry 0 rz 0.01 deg; joints [36.19, -46.806, 110.614, -140.977, 69.731, 165.244]
  MoveL 6337 to (-6.14, 73.39, -54.5) mm, rotated rx -180 ry 0 rz 0.01 deg; joints [36.225, -51.531, 121.474, -142.171, 74.547, 169.237]
  MoveC 6338 to (-4.01, 73.23, -54.5) mm, rotated rx 180 ry 0 rz 0.01 deg; joints [36.275, -51.595, 121.623, -142.135, 74.625, 169.277] to (-2.89, 75.05, -54.5) mm, rotated rx -180 ry 0 rz 0.01 deg; joints [36.369, -51.591, 121.608, -142.038, 74.637, 169.244]
  MoveL 6339 to (-2.9, 322.19, -54.5) mm, rotated rx -180 ry 0 rz 0.01 deg; joints [44.231, -45.702, 107.869, -132.463, 71.042, 161.231]
  MoveC 6340 to (-4.03, 324.91, -54.5) mm, rotated rx 180 ry 0 rz 0.01 deg; joints [44.277, -45.593, 107.624, -132.383, 70.966, 161.11] to (-6.75, 326.04, -54.5) mm, rotated rx -180 ry 0 rz 0.01 deg; joints [44.234, -45.481, 107.377, -132.391, 70.86, 161.019]
  MoveL 6341 to (-138.56, 326.04, -54.5) mm, rotated rx -180 ry 0 rz 0.01 deg; joints [40.849, -41.287, 98.25, -134.363, 66.221, 158.439]
  MoveC 6342 to (-140.5, 324.92, -54.5) mm, rotated rx -180 ry 0 rz 0.01 deg; joints [40.771, -41.253, 98.177, -134.43, 66.164, 158.442] to (-140.52, 322.68, -54.5) mm, rotated rx 180 ry 0 rz 0.01 deg; joints [40.709, -41.317, 98.319, -134.517, 66.194, 158.529]
  MoveC 6343 to (-138.94, 319.9, -54.5) mm, rotated rx 180 ry 0 rz 0.01 deg; joints [40.669, -41.451, 98.612, -134.607, 66.29, 158.669] to (-137.34, 317.13, -54.5) mm, rotated rx -180 ry 0 rz 0.01 deg; joints [40.629, -41.585, 98.905, -134.696, 66.387, 158.809]
  MoveC 6344 to (-135.98, 314.22, -54.5) mm, rotated rx -180 ry 0 rz 0.01 deg; joints [40.581, -41.714, 99.189, -134.794, 66.477, 158.949] to (-135.15, 311.12, -54.5) mm, rotated rx -180 ry 0 rz 0.01 deg; joints [40.514, -41.83, 99.445, -134.904, 66.55, 159.084]
  MoveC 6345 to (-134.26, 306.28, -54.5) mm, rotated rx 180 ry 0 rz 0.01 deg; joints [40.398, -41.997, 99.813, -135.082, 66.648, 159.287] to (-133.34, 301.44, -54.5) mm, rotated rx 180 ry 0 rz 0.01 deg; joints [40.283, -42.164, 100.182, -135.26, 66.748, 159.489]
  MoveC 6346 to (-132.5, 296.58, -54.5) mm, rotated rx -180 ry 0 rz 0.01 deg; joints [40.165, -42.328, 100.543, -135.439, 66.845, 159.689] to (-131.87, 291.69, -54.5) mm, rotated rx 180 ry 0 rz 0.01 deg; joints [40.04, -42.484, 100.89, -135.622, 66.935, 159.884]
  MoveL 6347 to (-119.75, 167.78, -54.5) mm, rotated rx -180 ry 0 rz 0.01 deg; joints [36.582, -46.029, 108.855, -140.341, 69.083, 164.433]
  MoveC 6348 to (-120.53, 163.96, -54.5) mm, rotated rx 180 ry 0 rz 0.01 deg; joints [36.442, -46.093, 109.002, -140.505, 69.107, 164.543] to (-123.32, 161.24, -54.5) mm, rotated rx 180 ry 0 rz 0.01 deg; joints [36.289, -46.064, 108.945, -140.655, 69.04, 164.581]
  MoveC 6349 to (-126.37, 159.02, -54.5) mm, rotated rx -180 ry 0 rz 0.01 deg; joints [36.147, -46.016, 108.842, -140.788, 68.957, 164.598] to (-128.59, 155.97, -54.5) mm, rotated rx -180 ry 0 rz 0.01 deg; joints [35.997, -46.014, 108.842, -140.942, 68.916, 164.657]
  MoveC 6350 to (-129.16, 154.94, -54.5) mm, rotated rx -180 ry 0 rz 0.01 deg; joints [35.951, -46.018, 108.855, -140.992, 68.908, 164.679] to (-129.82, 153.96, -54.5) mm, rotated rx 180 ry 0 rz 0.01 deg; joints [35.904, -46.019, 108.859, -141.041, 68.897, 164.699]
  MoveC 6351 to (-133.26, 149.82, -54.5) mm, rotated rx -180 ry 0 rz 0.01 deg; joints [35.691, -46.001, 108.825, -141.256, 68.825, 164.771] to (-137.2, 146.16, -54.5) mm, rotated rx 180 ry 0 rz 0.01 deg; joints [35.482, -45.954, 108.729, -141.459, 68.726, 164.817]
  MoveC 6352 to (-137.84, 145.66, -54.5) mm, rotated rx 180 ry 0 rz 0.01 deg; joints [35.451, -45.944, 108.708, -141.488, 68.709, 164.822] to (-138.5, 145.19, -54.5) mm, rotated rx -180 ry 0 rz 0.01 deg; joints [35.421, -45.933, 108.684, -141.516, 68.69, 164.825]
  MoveC 6353 to (-139.17, 144.74, -54.5) mm, rotated rx -180 ry 0 rz 0.01 deg; joints [35.391, -45.92, 108.658, -141.543, 68.671, 164.827] to (-139.87, 144.33, -54.5) mm, rotated rx 180 ry 0 rz 0.01 deg; joints [35.361, -45.907, 108.629, -141.57, 68.65, 164.828]
  MoveL 6354 to (-176.15, 123.35, -54.5) mm, rotated rx -180 ry 0 rz 0.01 deg; joints [33.87, -45.153, 107.008, -142.897, 67.54, 164.846]
  MoveC 6355 to (-181.6, 121.77, -54.5) mm, rotated rx -180 ry 0 rz 0.01 deg; joints [33.7, -45.001, 106.675, -143.028, 67.348, 164.798] to (-187.16, 122.91, -54.5) mm, rotated rx 180 ry 0 rz 0.01 deg; joints [33.617, -44.784, 106.196, -143.048, 67.115, 164.662]
  MoveC 6356 to (-191.63, 126.33, -54.5) mm, rotated rx -180 ry 0 rz 0.01 deg; joints [33.631, -44.552, 105.682, -142.961, 66.893, 164.471] to (-194.38, 131.24, -54.5) mm, rotated rx -180 ry 0 rz 0.01 deg; joints [33.731, -44.347, 105.222, -142.792, 66.719, 164.262]
  MoveC 6357 to (-194.69, 132.61, -54.5) mm, rotated rx 180 ry 0 rz 0.01 deg; joints [33.768, -44.305, 105.127, -142.739, 66.689, 164.212] to (-194.8, 134.02, -54.5) mm, rotated rx -180 ry 0 rz 0.01 deg; joints [33.811, -44.269, 105.047, -142.683, 66.666, 164.164]
  MoveL 6358 to (-194.21, 259.89, -54.5) mm, rotated rx 180 ry 0 rz 0.01 deg; joints [37.67, -41.181, 98.124, -137.587, 65.002, 159.793]
  MoveC 6359 to (-194.82, 261.38, -54.5) mm, rotated rx 180 ry 0 rz 0.01 deg; joints [37.7, -41.118, 97.987, -137.533, 64.958, 159.724] to (-196.32, 262, -54.5) mm, rotated rx 180 ry 0 rz 0.01 deg; joints [37.684, -41.047, 97.834, -137.523, 64.891, 159.669]
  MoveL 6360 to (-197.19, 262, -54.5) mm, rotated rx -180 ry 0 rz 0.01 deg; joints [37.665, -41.016, 97.766, -137.532, 64.857, 159.651]
  MoveC 6361 to (-198.69, 261.38, -54.5) mm, rotated rx 180 ry 0 rz 0.01 deg; joints [37.613, -40.979, 97.687, -137.571, 64.807, 159.643] to (-199.31, 259.89, -54.5) mm, rotated rx -180 ry 0 rz 0.01 deg; joints [37.556, -40.997, 97.728, -137.638, 64.803, 159.686]
  MoveL 6362 to (-198.71, 134.02, -54.5) mm, rotated rx 180 ry 0 rz 0.01 deg; joints [33.727, -44.132, 104.747, -142.728, 66.511, 164.093]
  MoveC 6363 to (-200.1, 128.5, -54.5) mm, rotated rx -180 ry 0 rz 0.01 deg; joints [33.521, -44.207, 104.922, -142.969, 66.529, 164.246] to (-203.93, 124.3, -54.5) mm, rotated rx 180 ry 0 rz 0.01 deg; joints [33.304, -44.166, 104.839, -143.184, 66.433, 164.311]
  MoveC 6364 to (-209.16, 122.21, -54.5) mm, rotated rx -180 ry 0 rz 0.01 deg; joints [33.127, -44.028, 104.541, -143.327, 66.252, 164.283] to (-214.79, 122.33, -54.5) mm, rotated rx 180 ry 0 rz 0.01 deg; joints [33.013, -43.825, 104.098, -143.382, 66.026, 164.175]
  MoveC 6365 to (-215.49, 122.53, -54.5) mm, rotated rx 180 ry 0 rz 0.01 deg; joints [33.004, -43.795, 104.033, -143.382, 65.995, 164.156] to (-216.18, 122.78, -54.5) mm, rotated rx 180 ry 0 rz 0.01 deg; joints [32.998, -43.765, 103.966, -143.379, 65.964, 164.135]
  MoveC 6366 to (-216.85, 123.08, -54.5) mm, rotated rx -180 ry 0 rz 0.01 deg; joints [32.994, -43.735, 103.899, -143.373, 65.933, 164.113] to (-217.5, 123.42, -54.5) mm, rotated rx 180 ry 0 rz 0.01 deg; joints [32.991, -43.704, 103.831, -143.366, 65.903, 164.089]
  MoveL 6367 to (-256.62, 146.38, -54.5) mm, rotated rx -180 ry 0 rz 0.01 deg; joints [32.915, -41.746, 99.537, -142.79, 64.011, 162.575]
  MoveC 6368 to (-260.34, 149.57, -54.5) mm, rotated rx -180 ry 0 rz 0.01 deg; joints [32.94, -41.531, 99.067, -142.689, 63.816, 162.391] to (-263.38, 153.42, -54.5) mm, rotated rx -180 ry 0 rz 0.01 deg; joints [32.998, -41.325, 98.615, -142.554, 63.64, 162.197]
  MoveC 6369 to (-265.52, 157.85, -54.5) mm, rotated rx 180 ry 0 rz 0.01 deg; joints [33.091, -41.139, 98.205, -142.387, 63.493, 162] to (-266.52, 162.67, -54.5) mm, rotated rx -180 ry 0 rz 0.01 deg; joints [33.22, -40.986, 97.867, -142.195, 63.389, 161.812]
  MoveC 6370 to (-266.54, 163.49, -54.5) mm, rotated rx 180 ry 0 rz 0.01 deg; joints [33.245, -40.965, 97.82, -142.161, 63.377, 161.782] to (-266.5, 164.32, -54.5) mm, rotated rx -180 ry 0 rz 0.01 deg; joints [33.271, -40.947, 97.779, -142.127, 63.368, 161.754]
  MoveL 6371 to (-252.26, 304.02, -54.5) mm, rotated rx -180 ry 0 rz 0.01 deg; joints [37.651, -37.765, 90.743, -136.259, 62.097, 156.777]
  MoveC 6372 to (-250.7, 309.42, -54.5) mm, rotated rx 180 ry 0 rz 0.01 deg; joints [37.834, -37.667, 90.525, -136.027, 62.088, 156.593] to (-248.52, 314.61, -54.5) mm, rotated rx -180 ry 0 rz 0.01 deg; joints [38.025, -37.598, 90.371, -135.8, 62.107, 156.432]
  MoveC 6373 to (-245.98, 319.61, -54.5) mm, rotated rx -180 ry 0 rz 0.01 deg; joints [38.218, -37.548, 90.257, -135.578, 62.142, 156.287] to (-243.29, 324.54, -54.5) mm, rotated rx 180 ry 0 rz 0.01 deg; joints [38.411, -37.505, 90.158, -135.359, 62.185, 156.148]
  MoveC 6374 to (-242.05, 326.34, -54.5) mm, rotated rx -180 ry 0 rz 0.01 deg; joints [38.488, -37.498, 90.142, -135.278, 62.21, 156.103] to (-240.52, 327.91, -54.5) mm, rotated rx -180 ry 0 rz 0.01 deg; joints [38.564, -37.51, 90.165, -135.204, 62.251, 156.075]
  MoveC 6375 to (-238.89, 329.35, -54.5) mm, rotated rx -180 ry 0 rz 0.01 deg; joints [38.639, -37.53, 90.205, -135.135, 62.297, 156.055] to (-237.28, 330.82, -54.5) mm, rotated rx 180 ry 0 rz 0.01 deg; joints [38.714, -37.548, 90.241, -135.065, 62.342, 156.032]
  MoveC 6376 to (-236.85, 332.74, -54.5) mm, rotated rx 180 ry 0 rz 0.01 deg; joints [38.776, -37.506, 90.15, -134.983, 62.334, 155.963] to (-238.48, 333.85, -54.5) mm, rotated rx 180 ry 0 rz 0.01 deg; joints [38.771, -37.41, 89.942, -134.948, 62.253, 155.877]
  MoveL 6377 to (-394.58, 333.84, -54.5) mm, rotated rx 180 ry 0 rz 0.01 deg; joints [35.593, -30.634, 75.665, -135.03, 55.466, 151.414]
  MoveC 6378 to (-397.3, 332.71, -54.5) mm, rotated rx -180 ry 0 rz 0.01 deg; joints [35.512, -30.539, 75.469, -135.066, 55.354, 151.376] to (-398.43, 329.99, -54.5) mm, rotated rx -180 ry 0 rz 0.01 deg; joints [35.419, -30.577, 75.552, -135.186, 55.339, 151.471]
  MoveL 6379 to (-398.42, 58.29, -54.5) mm, rotated rx -180 ry 0 rz 0.01 deg; joints [27.575, -38.023, 91.695, -147.265, 58.916, 162.695]
  MoveC 6380 to (-397.31, 56.66, -54.5) mm, rotated rx 180 ry 0 rz 0.01 deg; joints [27.542, -38.106, 91.876, -147.333, 58.987, 162.776] to (-395.39, 57.08, -54.5) mm, rotated rx -180 ry 0 rz 0.01 deg; joints [27.587, -38.18, 92.033, -147.31, 59.072, 162.802]
  MoveC 6381 to (-393.08, 59.4, -54.5) mm, rotated rx -180 ry 0 rz 0.01 deg; joints [27.697, -38.229, 92.134, -147.205, 59.15, 162.771] to (-390.64, 61.6, -54.5) mm, rotated rx -180 ry 0 rz 0.01 deg; joints [27.806, -38.286, 92.251, -147.105, 59.236, 162.747]
  MoveC 6382 to (-388.1, 63.67, -54.5) mm, rotated rx 180 ry 0 rz 0.01 deg; joints [27.913, -38.349, 92.383, -147.009, 59.328, 162.729] to (-385.48, 65.63, -54.5) mm, rotated rx 180 ry 0 rz 0.01 deg; joints [28.018, -38.418, 92.527, -146.917, 59.424, 162.716]
  MoveL 6383 to (-279.08, 142.21, -54.5) mm, rotated rx -180 ry 0 rz 0.01 deg; joints [32.339, -40.991, 97.915, -143.139, 63.131, 162.269]
  MoveC 6384 to (-274.2, 144.49, -54.5) mm, rotated rx 180 ry 0 rz 0.01 deg; joints [32.506, -41.125, 98.198, -143.008, 63.306, 162.288] to (-268.82, 144.86, -54.5) mm, rotated rx 180 ry 0 rz 0.01 deg; joints [32.624, -41.321, 98.622, -142.951, 63.526, 162.384]
  MoveC 6385 to (-263.59, 143.91, -54.5) mm, rotated rx 180 ry 0 rz 0.01 deg; joints [32.699, -41.542, 99.099, -142.949, 63.755, 162.521] to (-258.52, 142.31, -54.5) mm, rotated rx 180 ry 0 rz 0.01 deg; joints [32.75, -41.77, 99.595, -142.974, 63.985, 162.676]
  MoveC 6386 to (-257.67, 141.96, -54.5) mm, rotated rx 180 ry 0 rz 0.01 deg; joints [32.756, -41.81, 99.683, -142.982, 64.025, 162.705] to (-256.83, 141.55, -54.5) mm, rotated rx 180 ry 0 rz 0.01 deg; joints [32.761, -41.851, 99.771, -142.991, 64.065, 162.735]
  MoveC 6387 to (-256.01, 141.12, -54.5) mm, rotated rx 180 ry 0 rz 0.01 deg; joints [32.763, -41.891, 99.86, -143.002, 64.104, 162.766] to (-255.2, 140.67, -54.5) mm, rotated rx 180 ry 0 rz 0.01 deg; joints [32.766, -41.932, 99.95, -143.014, 64.144, 162.797]
  MoveL 6388 to (-219.43, 120.08, -54.5) mm, rotated rx -180 ry 0 rz 0.01 deg; joints [32.844, -43.709, 103.849, -143.523, 65.869, 164.162]
  MoveC 6389 to (-215.28, 116.09, -54.5) mm, rotated rx -180 ry 0 rz 0.01 deg; joints [32.802, -43.946, 104.373, -143.644, 66.088, 164.368] to (-213.46, 110.64, -54.5) mm, rotated rx -180 ry 0 rz 0.01 deg; joints [32.663, -44.13, 104.787, -143.849, 66.233, 164.576]
  MoveC 6390 to (-214.2, 104.97, -54.5) mm, rotated rx -180 ry 0 rz 0.01 deg; joints [32.464, -44.227, 105.01, -144.09, 66.277, 164.743] to (-217.18, 100.1, -54.5) mm, rotated rx 180 ry 0 rz 0.01 deg; joints [32.244, -44.227, 105.018, -144.323, 66.221, 164.844]
  MoveC 6391 to (-218.18, 99.19, -54.5) mm, rotated rx -180 ry 0 rz 0.01 deg; joints [32.194, -44.211, 104.985, -144.371, 66.193, 164.855] to (-219.3, 98.44, -54.5) mm, rotated rx -180 ry 0 rz 0.01 deg; joints [32.146, -44.187, 104.935, -144.414, 66.158, 164.858]
  MoveL 6392 to (-328.52, 36.08, -54.5) mm, rotated rx -180 ry 0 rz 0.01 deg; joints [28.043, -41.377, 98.942, -147.927, 62.344, 164.832]
  MoveC 6393 to (-329.5, 34.8, -54.5) mm, rotated rx 180 ry 0 rz 0.01 deg; joints [27.984, -41.364, 98.916, -147.987, 62.316, 164.855] to (-329.29, 33.19, -54.5) mm, rotated rx -180 ry 0 rz 0.01 deg; joints [27.935, -41.405, 99.007, -148.054, 62.345, 164.91]
  MoveL 6394 to (-328.85, 32.44, -54.5) mm, rotated rx 180 ry 0 rz 0.01 deg; joints [27.918, -41.437, 99.078, -148.083, 62.374, 164.942]
  MoveC 6395 to (-327.57, 31.45, -54.5) mm, rotated rx 180 ry 0 rz 0.01 deg; joints [27.908, -41.508, 99.233, -148.117, 62.442, 164.997] to (-325.97, 31.67, -54.5) mm, rotated rx -180 ry 0 rz 0.01 deg; joints [27.943, -41.567, 99.36, -148.098, 62.51, 165.02]
  MoveL 6396 to (-217.36, 95.08, -54.5) mm, rotated rx -180 ry 0 rz 0.01 deg; joints [32.076, -44.328, 105.251, -144.532, 66.28, 164.999]
  MoveC 6397 to (-211.85, 96.65, -54.5) mm, rotated rx 180 ry 0 rz 0.01 deg; joints [32.241, -44.49, 105.602, -144.407, 66.481, 165.049] to (-206.26, 95.45, -54.5) mm, rotated rx 180 ry 0 rz 0.01 deg; joints [32.317, -44.713, 106.094, -144.395, 66.721, 165.187]
  MoveC 6398 to (-201.78, 91.96, -54.5) mm, rotated rx -180 ry 0 rz 0.01 deg; joints [32.296, -44.945, 106.609, -144.488, 66.946, 165.375] to (-199.08, 86.97, -54.5) mm, rotated rx 180 ry 0 rz 0.01 deg; joints [32.187, -45.144, 107.058, -144.663, 67.119, 165.578]
  MoveC 6399 to (-198.79, 85.66, -54.5) mm, rotated rx 180 ry 0 rz 0.01 deg; joints [32.15, -45.182, 107.144, -144.714, 67.148, 165.623] to (-198.7, 84.31, -54.5) mm, rotated rx -180 ry 0 rz 0.01 deg; joints [32.107, -45.214, 107.216, -144.768, 67.17, 165.667]
  MoveL 6400 to (-199.06, 38.43, -54.5) mm, rotated rx 180 ry 0 rz 0.01 deg; joints [30.551, -46.128, 109.328, -146.675, 67.756, 167.038]
  MoveC 6401 to (-200.03, 33.61, -54.5) mm, rotated rx -180 ry 0 rz 0.01 deg; joints [30.366, -46.188, 109.472, -146.888, 67.78, 167.162] to (-201.93, 29.07, -54.5) mm, rotated rx -180 ry 0 rz 0.01 deg; joints [30.171, -46.21, 109.528, -147.099, 67.762, 167.262]
  MoveC 6402 to (-204.79, 25.06, -54.5) mm, rotated rx -180 ry 0 rz 0.01 deg; joints [29.976, -46.187, 109.487, -147.3, 67.699, 167.331] to (-208.54, 21.86, -54.5) mm, rotated rx -180 ry 0 rz 0.01 deg; joints [29.79, -46.117, 109.339, -147.477, 67.588, 167.361]
  MoveC 6403 to (-209.17, 21.47, -54.5) mm, rotated rx 180 ry 0 rz 0.01 deg; joints [29.765, -46.102, 109.306, -147.5, 67.567, 167.362] to (-209.83, 21.14, -54.5) mm, rotated rx -180 ry 0 rz 0.01 deg; joints [29.74, -46.086, 109.27, -147.522, 67.544, 167.36]
  MoveL 6404 to (-309.5, -23.25, -54.5) mm, rotated rx 180 ry 0 rz 0.01 deg; joints [26.391, -43.254, 103.134, -150.315, 63.892, 166.99]
  MoveC 6405 to (-310.29, -24.81, -54.5) mm, rotated rx -180 ry 0 rz 0.01 deg; joints [26.325, -43.252, 103.133, -150.387, 63.876, 167.023] to (-308.93, -25.91, -54.5) mm, rotated rx 180 ry 0 rz 0.01 deg; joints [26.31, -43.324, 103.292, -150.424, 63.948, 167.078]
  MoveL 6406 to (-84.59, -25.91, -54.5) mm, rotated rx 180 ry 0 rz 0.01 deg; joints [30.673, -51.043, 120.578, -147.769, 73.111, 170.632]
  MoveC 6407 to (-83.22, -24.81, -54.5) mm, rotated rx -180 ry 0 rz 0.01 deg; joints [30.745, -51.066, 120.628, -147.699, 73.147, 170.625] to (-84.01, -23.25, -54.5) mm, rotated rx 180 ry 0 rz 0.01 deg; joints [30.786, -51.015, 120.506, -147.646, 73.095, 170.573]
  MoveL 6408 to (-184.15, 21.4, -54.5) mm, rotated rx 180 ry 0 rz 0.01 deg; joints [30.264, -46.967, 111.229, -147.207, 68.577, 167.776]
  MoveC 6409 to (-188.27, 24.21, -54.5) mm, rotated rx 180 ry 0 rz 0.01 deg; joints [30.278, -46.773, 110.791, -147.14, 68.375, 167.628] to (-191.2, 28.24, -54.5) mm, rotated rx -180 ry 0 rz 0.01 deg; joints [30.359, -46.596, 110.388, -147.007, 68.205, 167.464]
  MoveC 6410 to (-193.07, 32.8, -54.5) mm, rotated rx -180 ry 0 rz 0.01 deg; joints [30.479, -46.444, 110.041, -146.839, 68.07, 167.301] to (-194.33, 37.56, -54.5) mm, rotated rx -180 ry 0 rz 0.01 deg; joints [30.617, -46.309, 109.73, -146.655, 67.958, 167.142]
  MoveC 6411 to (-194.67, 39.89, -54.5) mm, rotated rx -180 ry 0 rz 0.01 deg; joints [30.69, -46.252, 109.599, -146.563, 67.914, 167.069] to (-194.78, 42.23, -54.5) mm, rotated rx -180 ry 0 rz 0.01 deg; joints [30.768, -46.202, 109.484, -146.466, 67.878, 166.998]
  MoveL 6412 to (-194.81, 84.32, -54.5) mm, rotated rx -180 ry 0 rz 0.01 deg; joints [32.188, -45.349, 107.513, -144.723, 67.324, 165.734]
  MoveC 6413 to (-193.08, 90.61, -54.5) mm, rotated rx 180 ry 0 rz 0.01 deg; joints [32.433, -45.277, 107.343, -144.443, 67.31, 165.571] to (-188.35, 95.1, -54.5) mm, rotated rx -180 ry 0 rz 0.01 deg; joints [32.682, -45.345, 107.484, -144.202, 67.437, 165.515]
  MoveC 6414 to (-182.04, 96.63, -54.5) mm, rotated rx -180 ry 0 rz 0.01 deg; joints [32.867, -45.53, 107.889, -144.063, 67.666, 165.579] to (-175.78, 94.9, -54.5) mm, rotated rx 180 ry 0 rz 0.01 deg; joints [32.944, -45.781, 108.446, -144.056, 67.935, 165.742]
  MoveL 6415 to (-67.54, 31.67, -54.5) mm, rotated rx -180 ry 0 rz 0.01 deg; joints [33.195, -50.529, 119.256, -145.048, 72.935, 169.383]
  MoveC 6416 to (-65.94, 31.46, -54.5) mm, rotated rx -180 ry 0 rz 0.01 deg; joints [33.225, -50.581, 119.378, -145.029, 72.998, 169.415] to (-64.66, 32.44, -54.5) mm, rotated rx 180 ry 0 rz 0.01 deg; joints [33.291, -50.602, 119.422, -144.965, 73.032, 169.409]
  MoveL 6417 to (-64.22, 33.19, -54.5) mm, rotated rx -180 ry 0 rz 0.01 deg; joints [33.329, -50.601, 119.418, -144.926, 73.037, 169.396]
  MoveC 6418 to (-64.01, 34.8, -54.5) mm, rotated rx 180 ry 0 rz 0.01 deg; joints [33.392, -50.577, 119.36, -144.855, 73.022, 169.355] to (-65, 36.08, -54.5) mm, rotated rx -180 ry 0 rz 0.01 deg; joints [33.415, -50.523, 119.232, -144.819, 72.967, 169.304]
  MoveL 6419 to (-174.23, 98.45, -54.5) mm, rotated rx -180 ry 0 rz 0.01 deg; joints [33.095, -45.759, 108.39, -143.891, 67.948, 165.66]
  MoveC 6420 to (-178.43, 102.56, -54.5) mm, rotated rx -180 ry 0 rz 0.01 deg; joints [33.14, -45.527, 107.871, -143.775, 67.729, 165.459] to (-180.12, 108.19, -54.5) mm, rotated rx 180 ry 0 rz 0.01 deg; joints [33.289, -45.348, 107.466, -143.565, 67.587, 165.253]
  MoveC 6421 to (-179.12, 113.93, -54.5) mm, rotated rx 180 ry 0 rz 0.01 deg; joints [33.499, -45.258, 107.256, -143.318, 67.55, 165.091] to (-175.86, 118.75, -54.5) mm, rotated rx -180 ry 0 rz 0.01 deg; joints [33.727, -45.265, 107.261, -143.081, 67.613, 164.997]
  MoveC 6422 to (-175, 119.48, -54.5) mm, rotated rx -180 ry 0 rz 0.01 deg; joints [33.769, -45.278, 107.289, -143.04, 67.636, 164.99] to (-174.07, 120.09, -54.5) mm, rotated rx 180 ry 0 rz 0.01 deg; joints [33.81, -45.296, 107.328, -143.004, 67.665, 164.987]
  MoveL 6423 to (-133.77, 142.83, -54.5) mm, rotated rx -180 ry 0 rz 0.01 deg; joints [35.453, -46.142, 109.151, -141.545, 68.902, 164.985]
  MoveC 6424 to (-129.25, 144.31, -54.5) mm, rotated rx -180 ry 0 rz 0.01 deg; joints [35.605, -46.257, 109.403, -141.421, 69.051, 165.018] to (-124.53, 144.85, -54.5) mm, rotated rx -180 ry 0 rz 0.01 deg; joints [35.733, -46.399, 109.715, -141.33, 69.221, 165.084]
  MoveC 6425 to (-119.8, 144.36, -54.5) mm, rotated rx 180 ry 0 rz 0.01 deg; joints [35.828, -46.564, 110.082, -141.281, 69.405, 165.184] to (-115.32, 142.75, -54.5) mm, rotated rx 180 ry 0 rz 0.01 deg; joints [35.881, -46.745, 110.487, -141.279, 69.594, 165.314]
  MoveC 6426 to (-114.67, 142.4, -54.5) mm, rotated rx -180 ry 0 rz 0.01 deg; joints [35.884, -46.774, 110.552, -141.283, 69.623, 165.336] to (-114.06, 141.99, -54.5) mm, rotated rx 180 ry 0 rz 0.01 deg; joints [35.886, -46.803, 110.617, -141.291, 69.652, 165.36]
  MoveL 6427 to (-3.68, 62.27, -54.5) mm, rotated rx -180 ry 0 rz 0.01 deg; joints [35.891, -51.821, 122.173, -142.578, 74.802, 169.589]
  MoveC 6428 to (-2.23, 61.04, -54.5) mm, rotated rx -180 ry 0 rz 0.01 deg; joints [35.885, -51.886, 122.328, -142.6, 74.872, 169.647] to (-0.83, 59.75, -54.5) mm, rotated rx -180 ry 0 rz 0.01 deg; joints [35.874, -51.951, 122.482, -142.625, 74.941, 169.706]
  MoveC 6429 to (0.53, 58.43, -54.5) mm, rotated rx -180 ry 0 rz 0.01 deg; joints [35.862, -52.016, 122.635, -142.652, 75.009, 169.766] to (1.88, 57.09, -54.5) mm, rotated rx 180 ry 0 rz 0.01 deg; joints [35.849, -52.08, 122.788, -142.679, 75.077, 169.825]
  MoveC 6430 to (3.82, 56.72, -54.5) mm, rotated rx -180 ry 0 rz 0.01 deg; joints [35.886, -52.142, 122.934, -142.655, 75.151, 169.867] to (4.92, 58.36, -54.5) mm, rotated rx 180 ry 0 rz 0.01 deg; joints [35.975, -52.141, 122.928, -142.565, 75.165, 169.84]
  MoveL 6431 to (4.91, 330, -54.5) mm, rotated rx 180 ry 0 rz 0.01 deg; joints [44.666, -45.712, 107.879, -132.032, 71.192, 161.087]
  MoveC 6432 to (3.78, 332.72, -54.5) mm, rotated rx -180 ry 0 rz 0.01 deg; joints [44.711, -45.603, 107.634, -131.953, 71.117, 160.966] to (1.06, 333.85, -54.5) mm, rotated rx 180 ry 0 rz 0.01 deg; joints [44.667, -45.491, 107.387, -131.961, 71.011, 160.874]
  MoveL 6433 to (-155.02, 333.85, -54.5) mm, rotated rx 180 ry 0 rz 0.01 deg; joints [40.672, -40.488, 96.52, -134.243, 65.501, 157.784]
  MoveC 6434 to (-156.65, 332.74, -54.5) mm, rotated rx -180 ry 0 rz 0.01 deg; joints [40.603, -40.464, 96.469, -134.304, 65.454, 157.792] to (-156.22, 330.82, -54.5) mm, rotated rx 180 ry 0 rz 0.01 deg; joints [40.56, -40.535, 96.625, -134.375, 65.497, 157.878]
  MoveC 6435 to (-154.62, 329.34, -54.5) mm, rotated rx -180 ry 0 rz 0.01 deg; joints [40.557, -40.635, 96.841, -134.415, 65.577, 157.97] to (-152.98, 327.91, -54.5) mm, rotated rx -180 ry 0 rz 0.01 deg; joints [40.556, -40.734, 97.056, -134.454, 65.658, 158.061]
  MoveC 6436 to (-151.46, 326.34, -54.5) mm, rotated rx -180 ry 0 rz 0.01 deg; joints [40.549, -40.832, 97.271, -134.499, 65.736, 158.155] to (-150.23, 324.54, -54.5) mm, rotated rx -180 ry 0 rz 0.01 deg; joints [40.528, -40.928, 97.478, -134.556, 65.807, 158.252]
  MoveC 6437 to (-147.84, 320.23, -54.5) mm, rotated rx 180 ry 0 rz 0.01 deg; joints [40.465, -41.135, 97.93, -134.698, 65.954, 158.47] to (-145.54, 315.88, -54.5) mm, rotated rx -180 ry 0 rz 0.01 deg; joints [40.398, -41.339, 98.378, -134.842, 66.099, 158.687]
  MoveC 6438 to (-143.48, 311.4, -54.5) mm, rotated rx 180 ry 0 rz 0.01 deg; joints [40.321, -41.537, 98.812, -134.993, 66.237, 158.902] to (-141.87, 306.74, -54.5) mm, rotated rx 180 ry 0 rz 0.01 deg; joints [40.228, -41.725, 99.223, -135.156, 66.36, 159.113]
  MoveC 6439 to (-140.94, 302.83, -54.5) mm, rotated rx 180 ry 0 rz 0.01 deg; joints [40.14, -41.866, 99.536, -135.298, 66.447, 159.281] to (-140.41, 298.85, -54.5) mm, rotated rx 180 ry 0 rz 0.01 deg; joints [40.04, -41.996, 99.822, -135.448, 66.521, 159.443]
  MoveC 6440 to (-140.04, 294.85, -54.5) mm, rotated rx -180 ry 0 rz 0.01 deg; joints [39.934, -42.12, 100.096, -135.6, 66.589, 159.601] to (-139.64, 290.86, -54.5) mm, rotated rx 180 ry 0 rz 0.01 deg; joints [39.83, -42.244, 100.371, -135.751, 66.658, 159.759]
  MoveL 6441 to (-127.01, 164.32, -54.5) mm, rotated rx -180 ry 0 rz 0.01 deg; joints [36.301, -45.873, 108.516, -140.585, 68.86, 164.415]
  MoveC 6442 to (-127.2, 160.03, -54.5) mm, rotated rx -180 ry 0 rz 0.01 deg; joints [36.16, -45.966, 108.729, -140.759, 68.912, 164.55] to (-128.59, 155.97, -54.5) mm, rotated rx 180 ry 0 rz 0.01 deg; joints [35.997, -46.014, 108.842, -140.942, 68.916, 164.657]
  MoveL 6443 to (-128.72, 155.36, -54.33) mm, rotated rx 180 ry 0 rz 0.01 deg; joints [35.974, -46.033, 108.866, -140.967, 68.913, 164.668]
  MoveL 6444 to (-128.62, 154.9, -53.87) mm, rotated rx -180 ry 0 rz 0.01 deg; joints [35.962, -46.072, 108.9, -140.978, 68.905, 164.669]
  MoveL 6445 to (-128.54, 154.75, -53.23) mm, rotated rx -180 ry 0 rz 0.01 deg; joints [35.958, -46.113, 108.917, -140.976, 68.886, 164.655]
  Set speed (500.0 mm/s)
  MoveL 6446 to (-128.54, 154.75, 11) mm, rotated rx 180 ry 0 rz 0.01 deg; joints [35.925, -49.589, 109.146, -140.161, 66.366, 162.437]
  Set speed (500.0 mm/s)
  MoveL 6447 to (0.37, 325.79, 11) mm, rotated rx -180 ry 0 rz 0.01 deg; joints [44.397, -49.206, 108.086, -131.406, 68.906, 158.571]
  Set speed (100.0 mm/s)
  MoveL 6448 to (0.37, 325.79, -32.73) mm, rotated rx 180 ry 0 rz 0.01 deg; joints [44.414, -46.881, 107.97, -132.002, 70.382, 160.324]
  MoveL 6449 to (0.25, 325.89, -33.35) mm, rotated rx 180 ry 0 rz 0.01 deg; joints [44.414, -46.841, 107.953, -132.008, 70.397, 160.342]
  MoveL 6450 to (-0.08, 326.19, -33.82) mm, rotated rx 180 ry 0 rz 0.01 deg; joints [44.413, -46.797, 107.91, -132.009, 70.397, 160.343]
  MoveL 6451 to (-0.5, 326.64, -34) mm, rotated rx 180 ry 0 rz 0.01 deg; joints [44.415, -46.762, 107.854, -132.002, 70.384, 160.326]
  MoveL 6452 to (-1.23, 333.21, -34.24) mm, rotated rx -180 ry 0 rz 0.01 deg; joints [44.579, -46.538, 107.39, -131.776, 70.283, 160.08]
  MoveL 6453 to (4.49, 336.51, -34.49) mm, rotated rx -180 ry 0 rz 0.01 deg; joints [44.829, -46.6, 107.547, -131.554, 70.436, 160.069]
  MoveL 6454 to (9.81, 332.59, -34.73) mm, rotated rx 180 ry 0 rz 0.01 deg; joints [44.867, -46.858, 108.135, -131.603, 70.67, 160.318]
  MoveL 6455 to (8.35, 326.15, -34.98) mm, rotated rx -180 ry 0 rz 0.01 deg; joints [44.646, -46.987, 108.449, -131.87, 70.714, 160.539]
  MoveL 6456 to (1.86, 324.91, -35.22) mm, rotated rx 180 ry 0 rz 0.01 deg; joints [44.431, -46.816, 108.11, -132.039, 70.525, 160.48]
  MoveL 6457 to (-1.88, 330.35, -35.46) mm, rotated rx 180 ry 0 rz 0.01 deg; joints [44.481, -46.535, 107.524, -131.909, 70.339, 160.222]
  MoveL 6458 to (1.61, 335.96, -35.71) mm, rotated rx 180 ry 0 rz 0.01 deg; joints [44.734, -46.465, 107.391, -131.642, 70.389, 160.085]
  MoveL 6459 to (8.15, 335.01, -35.95) mm, rotated rx -180 ry 0 rz 0.01 deg; joints [44.889, -46.674, 107.87, -131.56, 70.624, 160.247]
  MoveL 6460 to (9.9, 328.64, -36.2) mm, rotated rx -180 ry 0 rz 0.01 deg; joints [44.759, -46.895, 108.385, -131.765, 70.773, 160.523]
  MoveL 6461 to (4.76, 324.49, -36.44) mm, rotated rx -180 ry 0 rz 0.01 deg; joints [44.5, -46.848, 108.317, -132.016, 70.667, 160.594]
  MoveL 6462 to (-1.1, 327.52, -36.68) mm, rotated rx -180 ry 0 rz 0.01 deg; joints [44.424, -46.573, 107.747, -132.015, 70.442, 160.387]
  MoveL 6463 to (-0.67, 334.11, -36.93) mm, rotated rx 180 ry 0 rz 0.01 deg; joints [44.62, -46.384, 107.356, -131.766, 70.378, 160.16]
  MoveL 6464 to (5.54, 336.36, -37.17) mm, rotated rx -180 ry 0 rz 0.01 deg; joints [44.855, -46.492, 107.611, -131.574, 70.561, 160.198]
  MoveL 6465 to (10.09, 331.56, -37.42) mm, rotated rx 180 ry 0 rz 0.01 deg; joints [44.847, -46.751, 108.206, -131.669, 70.781, 160.466]
  MoveL 6466 to (7.52, 325.48, -37.66) mm, rotated rx 180 ry 0 rz 0.01 deg; joints [44.605, -46.835, 108.425, -131.944, 70.785, 160.654]
  MoveL 6467 to (0.92, 325.4, -37.9) mm, rotated rx 180 ry 0 rz 0.01 deg; joints [44.42, -46.628, 108.005, -132.072, 70.577, 160.549]
  MoveL 6468 to (-1.81, 331.41, -38.15) mm, rotated rx 180 ry 0 rz 0.01 deg; joints [44.514, -46.362, 107.448, -131.902, 70.415, 160.287]
  MoveL 6469 to (2.61, 336.32, -38.39) mm, rotated rx -180 ry 0 rz 0.01 deg; joints [44.773, -46.34, 107.42, -131.644, 70.505, 160.194]
  MoveL 6470 to (8.88, 334.23, -38.64) mm, rotated rx -180 ry 0 rz 0.01 deg; joints [44.889, -46.572, 107.953, -131.609, 70.746, 160.393]
  MoveL 6471 to (9.48, 327.66, -38.88) mm, rotated rx -180 ry 0 rz 0.01 deg; joints [44.721, -46.765, 108.407, -131.843, 70.861, 160.656]
